(* CODESYS project pp-csp-handover-v4.project

Project tree, tasks and I/O mapping:
  PLC : HX-CP1S08, Hitachi Industrial Equipment Systems Co., Ltd., order no. HX-CP1S08, version 3.5.8.24
      settings: IP Address = '192.168.137.20'
    application Application
      libraries: Unit Conversion Interfaces, * (Intern); Standard, * (System); VisuDialogs, * (System); CAA Device Diagnosis, 3.5.4.0 (CAA Technical Workgroup); CAA Net Base Services, 3.5.8.10 (CAA Technical Workgroup); NetVarUdp, 3.5.17.0 (System); PRO JSON, 1.0.0.13 (Pro Electric)
      task VISU_TASK (cyclic, interval 200 ms, priority 31) calls VisuElems.Visu_Prg
      task EtherCAT_Task (cyclic, interval 4 ms, priority 1) calls CSP_Cycle, CSP_WriteOutputs
      task Task (cyclic, interval 5 ms, priority 5) calls main, TcpClient
      global variables gvlSetting
      data type ServoData
      program TcpClient [ST]
      program main [ST]
      visualisation Main
      global variables GVL
      program DriveDiagnostics [ST]
      function AppendDiagnosticText [ST]
      function BuildDiagnosticFeedback [ST]
      function LongStringLength [ST]
      data type CSP_AxisData
      function CSP_Bezier [ST]
      function block CSP_Brake [ST]
      global variables CSP_Config
      program CSP_Cycle [ST]
      global variables CSP_Data
      function CSP_Feedback [ST]
      function CSP_ParseFrame [ST]
      function CSP_ReadAxis [ST]
      function CSP_ReadNumber [ST]
      function block CSP_Receive [ST]
      function block CSP_Trajectory6 [ST]
      function CSP_WriteAxis [ST]
      program CSP_WriteOutputs [ST]
      data type PlatformControlState
      program PlatformStartup [ST]
      function CSP_StopOffset [ST]
    Basic : Basic, Hitachi-IES, version 3.5.8.20
      _16_Digital_Input : 16 Digital Input, Hitachi-IES, version 3.4.0.0
          input  Application.GVL.resetButton : BOOL  // ReserveWord0Type.Bit1
          input  Application.GVL.startButton : BOOL  // ReserveWord0Type.Bit2
          input  Application.GVL.stopButton : BOOL  // ReserveWord0Type.Bit3
          input  Application.GVL.safetySystem : BOOL  // ReserveWord0Type.Bit4
          unmapped channels: ReserveWord0Type, ReserveWord0Type, ReserveWord0Type
      _16_Digital_Output : 16 Digital Output, Hitachi-IES, version 3.4.0.0
          output Application.GVL.LightGreen : BOOL  // ReserveWord0Type.Bit0
          output Application.GVL.LightYellow : BOOL  // ReserveWord0Type.Bit1
          output Application.GVL.LightRed : BOOL  // ReserveWord0Type.Bit2
          unmapped channels: ReserveWord0Type, ReserveWord0Type, ReserveWord0Type
      <Empty>
      <Empty>
      _16_Digital_Input_1 : 16 Digital Input, Hitachi-IES, version 3.4.0.0
          unmapped channels: ReserveWord0Type, ReserveWord0Type, ReserveWord0Type
      <Empty>
      <Empty>
      <Empty>
      <Empty>
      <Empty>
      _16_Digital_Output_1 : 16 Digital Output, Hitachi-IES, version 3.4.0.0
          unmapped channels: ReserveWord0Type, ReserveWord0Type, ReserveWord0Type
    EtherCAT_Master : EtherCAT Master, Festo, version 3.5.16.43
        settings: MasterCycleTime = 4000; MasterUseLRW = False; SlaveAutoRestart = True; NetworkName = 'eth2'; NetworkName = "eth2"; SelectNetworkByName = False; EnableTaskMessage = False; SrcAddress1 = 42135; SrcAddress2 = 3137775364; EnableSecondAdapter = False; SrcAddress = [16#A4,16#97,16#BB,16#06,16#A7,16#04]; NetworkName = 'eth2'; NetworkName = "eth2"; SelectNetworkByName = False
      servo_drive_4 : CMMT-AS (FlightSim PP/CSP), Festo, order no. 5340819, 534082x, 813335x, version 1.0.0.0
          settings: Watchdog register 0400 = 2498; Watchdog register 0410 = 3000; Watchdog register 0420 = 1000; Physical Address of the Slave = 1002; AutoIncr Address of the Slave = 4294967295; FMMU.Global Start Address = 16#02000018; FMMU.Physical Start Address = 16#1000; FMMU.Access = 16#02; FMMU.Global Start Address = 16#01000012; FMMU.Physical Start Address = 16#1100; FMMU.Access = 16#01; FMMU.Global Start Address = 16#00080000; FMMU.StartBit = 1; FMMU.EndBit = 1; FMMU.Physical Start Address = 16#080D; FMMU.Access = 16#01; DC sync0 cycletime = 4000; DC enable = 1; DC sync0 enable = 1; DC sync1 cycletime = 4000; DC sync1 enable = 0
          unmapped channels: Controlword, Modes of operation, Target position, Profile velocity, Target velocity, Target torque, Velocity offset, Torque offset, ---, Statusword, Modes of operation display, Position actual value, Velocity actual value, Torque actual value, Multiturns actual value, ---
      servo_drive_3 : CMMT-AS (FlightSim PP/CSP), Festo, order no. 5340819, 534082x, 813335x, version 1.0.0.0
          settings: Watchdog register 0400 = 2498; Watchdog register 0410 = 3000; Watchdog register 0420 = 1000; Physical Address of the Slave = 1002; AutoIncr Address of the Slave = 4294967295; FMMU.Global Start Address = 16#02000018; FMMU.Physical Start Address = 16#1000; FMMU.Access = 16#02; FMMU.Global Start Address = 16#01000012; FMMU.Physical Start Address = 16#1100; FMMU.Access = 16#01; FMMU.Global Start Address = 16#00080000; FMMU.StartBit = 1; FMMU.EndBit = 1; FMMU.Physical Start Address = 16#080D; FMMU.Access = 16#01; DC sync0 cycletime = 4000; DC enable = 1; DC sync0 enable = 1; DC sync1 cycletime = 4000; DC sync1 enable = 0
          unmapped channels: Controlword, Modes of operation, Target position, Profile velocity, Target velocity, Target torque, Velocity offset, Torque offset, ---, Statusword, Modes of operation display, Position actual value, Velocity actual value, Torque actual value, Multiturns actual value, ---
      servo_drive_2 : CMMT-AS (FlightSim PP/CSP), Festo, order no. 5340819, 534082x, 813335x, version 1.0.0.0
          settings: Watchdog register 0400 = 2498; Watchdog register 0410 = 3000; Watchdog register 0420 = 1000; Physical Address of the Slave = 1002; AutoIncr Address of the Slave = 4294967295; FMMU.Global Start Address = 16#02000018; FMMU.Physical Start Address = 16#1000; FMMU.Access = 16#02; FMMU.Global Start Address = 16#01000012; FMMU.Physical Start Address = 16#1100; FMMU.Access = 16#01; FMMU.Global Start Address = 16#00080000; FMMU.StartBit = 1; FMMU.EndBit = 1; FMMU.Physical Start Address = 16#080D; FMMU.Access = 16#01; DC sync0 cycletime = 4000; DC enable = 1; DC sync0 enable = 1; DC sync1 cycletime = 4000; DC sync1 enable = 0
          unmapped channels: Controlword, Modes of operation, Target position, Profile velocity, Target velocity, Target torque, Velocity offset, Torque offset, ---, Statusword, Modes of operation display, Position actual value, Velocity actual value, Torque actual value, Multiturns actual value, ---
      servo_drive_1 : CMMT-AS (FlightSim PP/CSP), Festo, order no. 5340819, 534082x, 813335x, version 1.0.0.0
          settings: Watchdog register 0400 = 2498; Watchdog register 0410 = 3000; Watchdog register 0420 = 1000; Physical Address of the Slave = 1001; FMMU.Global Start Address = 16#02000000; FMMU.Physical Start Address = 16#1000; FMMU.Access = 16#02; FMMU.Global Start Address = 16#01000000; FMMU.Physical Start Address = 16#1100; FMMU.Access = 16#01; FMMU.Global Start Address = 16#00080000; FMMU.Physical Start Address = 16#080D; FMMU.Access = 16#01; DC sync0 cycletime = 4000; DC enable = 1; DC sync0 enable = 1; DC sync1 cycletime = 4000; DC sync1 enable = 0
          unmapped channels: Controlword, Modes of operation, Target position, Profile velocity, Target velocity, Target torque, Velocity offset, Torque offset, ---, Statusword, Modes of operation display, Position actual value, Velocity actual value, Torque actual value, Multiturns actual value, ---
      servo_drive_6 : CMMT-AS (FlightSim PP/CSP), Festo, order no. 5340819, 534082x, 813335x, version 1.0.0.0
          settings: Watchdog register 0400 = 2498; Watchdog register 0410 = 3000; Watchdog register 0420 = 1000; Physical Address of the Slave = 1002; AutoIncr Address of the Slave = 4294967295; FMMU.Global Start Address = 16#02000018; FMMU.Physical Start Address = 16#1000; FMMU.Access = 16#02; FMMU.Global Start Address = 16#01000012; FMMU.Physical Start Address = 16#1100; FMMU.Access = 16#01; FMMU.Global Start Address = 16#00080000; FMMU.StartBit = 1; FMMU.EndBit = 1; FMMU.Physical Start Address = 16#080D; FMMU.Access = 16#01; DC sync0 cycletime = 4000; DC enable = 1; DC sync0 enable = 1; DC sync1 cycletime = 4000; DC sync1 enable = 0
          unmapped channels: Controlword, Modes of operation, Target position, Profile velocity, Target velocity, Target torque, Velocity offset, Torque offset, ---, Statusword, Modes of operation display, Position actual value, Velocity actual value, Torque actual value, Multiturns actual value, ---
      servo_drive_5 : CMMT-AS (FlightSim PP/CSP), Festo, order no. 5340819, 534082x, 813335x, version 1.0.0.0
          settings: Watchdog register 0400 = 2498; Watchdog register 0410 = 3000; Watchdog register 0420 = 1000; Physical Address of the Slave = 1002; AutoIncr Address of the Slave = 4294967295; FMMU.Global Start Address = 16#02000018; FMMU.Physical Start Address = 16#1000; FMMU.Access = 16#02; FMMU.Global Start Address = 16#01000012; FMMU.Physical Start Address = 16#1100; FMMU.Access = 16#01; FMMU.Global Start Address = 16#00080000; FMMU.StartBit = 1; FMMU.EndBit = 1; FMMU.Physical Start Address = 16#080D; FMMU.Access = 16#01; DC sync0 cycletime = 4000; DC enable = 1; DC sync0 enable = 1; DC sync1 cycletime = 4000; DC sync1 enable = 0
          unmapped channels: Controlword, Modes of operation, Target position, Profile velocity, Target velocity, Target torque, Velocity offset, Torque offset, ---, Statusword, Modes of operation display, Position actual value, Velocity actual value, Torque actual value, Multiturns actual value, ---
  libraries: VisuSymbols, 4.1.0.0 (System)
  function block Axis [ST]: enabled, init, doAbort, isReady, doMovement, doReset, getPosition, inError, cycle, isInitialised, PPMoveDone
  function block signal [ST]: init, cycle
  text list GlobalTextList
  function block Light [ST]: blink, init, cycle, enable
  function block FlightSimulator [ST]: safetyStop, doReset, isEnabled, getPositions, cycle, goNeutralPosition, isReady, doMovement, isInitialised, init, inError, goHomePosition, goTopPosition, PPState
  data type stateFlightSimulator
*)

// PLC/Application/ServoData
TYPE ServoData :
STRUCT
	positions: ARRAY[1..6] OF JSONVAR;
	speeds: ARRAY[1..6] OF JSONVAR;
END_STRUCT
END_TYPE

// stateFlightSimulator
{attribute 'qualified_only'}
{attribute 'strict'}
TYPE stateFlightSimulator :
(
	error  := 0,
	resetting,
	stopped,
	starting,
	started,
	stopping
);
END_TYPE

// PLC/Application/CSP_AxisData
TYPE CSP_AxisData :
STRUCT
    RequestedPosition : LREAL;
    CommandPosition : LREAL;
    CommandVelocity : LREAL;
    CommandAcceleration : LREAL;
    ActualPosition : LREAL;
    ActualVelocity : LREAL;
    FollowingError : LREAL;
    PositionFactor : LREAL;
    VelocityFactor : LREAL;
    ActualRaw : DINT;
    TargetRaw : DINT;
    FollowingErrorRaw : DINT;
    ModeRequested : SINT;
    ModeActual : SINT;
    Statusword : WORD;
    Controlword : WORD;
    CiA402State : WORD;
    PositionLimit : BOOL;
    CommunicationTimeout : BOOL;
    Ready : BOOL;
    // 0 ready; 1 PDO pointer; 2 SDO init; 3 factor; 4 bus; 5 conversion mismatch.
    ReadinessCode : UINT;
    VelocityAllowed : LREAL;
END_STRUCT
END_TYPE

// PLC/Application/PlatformControlState
{attribute 'qualified_only'}
{attribute 'strict'}
TYPE PlatformControlState :
(
    PP_RESET := 0,
    PP_STOPPED := 1,
    PP_STARTING := 2,
    CSP_HANDOVER := 3,
    CSP_READY := 4,
    CSP_RUNNING := 5,
    CSP_RECOVERY := 6,
    FAULT := 7,
    PP_HANDBACK := 8 // Reset: CSP brakes and restores mode 1, then PP resumes
);
END_TYPE

// PLC/Application/gvlSetting
{attribute 'qualified_only'}
VAR_GLOBAL CONSTANT
    // Port to use to send data.
	gc_uiPort        : UINT := 32760;
    // IP Address of the computer that hosts the software.
	gc_stIpAddr      : NBS.IP_ADDR := (sAddr := '192.168.137.123');
	// Length of the telegram.
    gc_wMaxTelegram  : INT := 512;
END_VAR

// PLC/Application/GVL
{attribute 'qualified_only'}
VAR_GLOBAL
	// Red light on electrical housing.
	lightRed: BOOL;
	// Yellow light on electrical housing.
	lightYellow: BOOL;
	// Green light on electrical housing.
	lightGreen: BOOL;
	// Reset button on electrical housing.
	resetButton: BOOL := FALSE;
	// Start button on electrical housing.
	startButton: BOOL := FALSE;
	// Stop button on electrical housing.
	stopButton: BOOL := FALSE;
	// Safety system, connected to safety relay.
	safetySystem: BOOL := FALSE;
	// Virtual reset button on HMI.
	resetHMI: BOOL;
	// Virtual start button on HMI.
	startHMI: BOOL;
	// Virtual stop button on HMI.
	stopHMI: BOOL;
	// Virtual toggle button to toggle between tCP data and manual data on HMI.
	useTCPData: BOOL := TRUE;
	// Manual slider velocity input on HMI.
	nextVelocityInput: REAL := 200;
	// Manual slider position input on HMI.
	nextPositionInput: REAL := 0;
	// Flight simulator object.
	FlightSimulator: FlightSimulator;
	// Velocity input from TCP data or HMI data.
	servoVelocities: ARRAY[1..6] OF REAL;
	// Position input from TCP data or HMI data.
	servoPositions: ARRAY[1..6] OF REAL;
	// Current Positions in array format.
	servoPositionsCurrent: ARRAY[1..6] OF REAL;
	// Current Positions in JSON format, used to send back to TCP client.
	currentPositions: ARRAY[1..6] OF JSONVAR;
END_VAR

// PLC/Application/CSP_Config
{attribute 'qualified_only'}
VAR_GLOBAL CONSTANT
    CONTROL_MODE_PP : SINT := 1;
    CONTROL_MODE_CSP : SINT := 8;
    // Match BuildMode.h. PP remains the initial commissioning selection.
    ControlMode : SINT := 8;
    // Also set EtherCAT_Task, master cycle and slave DC Sync0 to this interval.
    CycleSeconds : LREAL := 0.004;
    MinimumPosition : LREAL := 10.0;
    MaximumPosition : LREAL := 390.0;
    MaximumVelocity : LREAL := 100; // mm/s; commissioning starting values
    MaximumAcceleration : LREAL := 200; // mm/s^2
    BrakingAcceleration : LREAL := 200; // <= MaximumAcceleration
    MaximumJerk : LREAL := 1000; // mm/s^3
    CommunicationTimeout : TIME := T#500MS;
    TransitionTimeout : TIME := T#10S;
    StandstillVelocity : LREAL := 0.05;
    HomePosition : LREAL := 200.0;
    HomeTolerance : LREAL := 0.5;
    HomeSettleTime : TIME := T#200MS;
    HomeTimeout : TIME := T#60S;
    // Set TRUE only after the eight required PDOs, DC, interpolation period,
    // actual task timing and all six existing position conversions are checked.
    Commissioned : BOOL := TRUE;
END_VAR

// PLC/Application/CSP_Data
{attribute 'qualified_only'}
VAR_GLOBAL
    Axis : ARRAY[1..6] OF CSP_AxisData;
    CycleCounter : UDINT;
    // TCP writes odd generation, complete target, then even generation. The
    // higher-priority motion task only accepts matching even generations.
    Generation : UDINT;
    ReceivedPosition : ARRAY[1..6] OF LREAL;
    ReceivedMode : SINT;
    ReceivedTick : UDINT;
    Connected : BOOL;
    Enable : BOOL;
    Reset : BOOL;
    StopRequested : BOOL;
    ResetRequired : BOOL := TRUE;
    Homing : BOOL; // park at HomePosition using the existing encoder reference
    ReadyToStart : BOOL;
    OwnsOutputs : BOOL; // FALSE: vendor PP writer; TRUE: direct CSP writer
    PlatformState : PlatformControlState := PlatformControlState.PP_RESET;
    PPReleased : BOOL; // published by PP task only after its last complete call
    // Published by the CSP task only after it restored mode 1 and stopped writing.
    // PP clears PPReleased in response; CSP then clears this flag.
    CSPReleased : BOOL;
    PPMoveDone : ARRAY[1..6] OF BOOL;
    AllPPMoveDone, AllStationary, AllCSPModeConfirmed : BOOL;
    // The exact PP-side handover condition, evaluated in the PP task.
    PPStartupComplete : BOOL;
    // First axis whose mode display differs from the requested handover mode
    // (8 during CSP_HANDOVER, 1 during PP_HANDBACK); 0 = all confirmed.
    ModeBlockingAxis : INT;
    InitialTargetRaw : ARRAY[1..6] OF DINT;
    // FaultCode that Reset acknowledged before ownership returned to PP.
    LastCSPFaultCode : UINT;
    Active : BOOL;
    TransitionState : UINT;
    Fault : BOOL;
    FaultCode : UINT;
    // Frozen at timeout, before quick stop changes the live drive states.
    TimeoutState : UINT;
    TimeoutStatusword : ARRAY[1..6] OF WORD;
    TimeoutControlword : ARRAY[1..6] OF WORD;
    // 0 running/transitioning; 1 commissioning; 2 axis readiness; 3 safety;
    // 4 operator Start; 5 fresh PC target; 6 drive mode; 7 fault (see FaultCode).
    // While PP owns the drives: 10 PP not in STARTED; 11 not stationary;
    // 12 PP move still executing / no drive Standstill (FlightSimulator.isReady);
    // 13 an axis is outside HomeTolerance of HomePosition; 14 MC_MoveAbsolute
    // Error/CommandAborted. PPMoveDone[1..6] shows the axis.
    StartupBlockReason : UINT;
    ReversalDeferred : BOOL;
    // Map 0x60F4:00 (DINT) from each drive here; not computed PC error.
    FollowingErrorRaw : ARRAY[1..6] OF DINT;
END_VAR

// PLC/Application/CSP_Cycle
PROGRAM CSP_Cycle
VAR
    trajectory : CSP_Trajectory6;
    actual, requested, receivedCopy : ARRAY[1..6] OF LREAL;
    generation, generationAfter, acceptedGeneration, tick : UDINT;
    packetMode : SINT;
    packetTick, receivedTickCopy : UDINT;
    newTarget, timedOut, allReady, allStopped, allDisabled, allMode, allEnabled, allSwitchedOn, allPPMode : BOOL;
    resetEdge : R_TRIG;
    resetRequest : BOOL;
    resetConditionsReady, anyDriveFaultReaction : BOOL;
    standstill : TON;
    transition : TON;
    previousTransitionState : UINT;
    homePhase : UINT; // 1 brake, 2 plan park move, 3 wait for measured arrival
    homeTarget : ARRAY[1..6] OF LREAL;
    homeSettled, homeTimer : TON;
    homeAtPosition : BOOL;
    handoverValid : BOOL;
    initialPosition : ARRAY[1..6] OF LREAL; // captured at the PP -> CSP ownership switch
    holdRaw : ARRAY[1..6] OF DINT; // stationary target while restoring PP mode
    expectedMode : SINT;
    i : INT;
    stateWord : WORD;
    distance : LREAL;
END_VAR

IF CSP_Config.ControlMode <> CSP_Config.CONTROL_MODE_CSP THEN RETURN; END_IF
CSP_Data.CycleCounter := CSP_Data.CycleCounter+1;
CSP_ReadAxis(Axis:=servo_drive_1,PlatformAxis:=1);
CSP_ReadAxis(Axis:=servo_drive_2,PlatformAxis:=2);
CSP_ReadAxis(Axis:=servo_drive_3,PlatformAxis:=3);
CSP_ReadAxis(Axis:=servo_drive_4,PlatformAxis:=4);
CSP_ReadAxis(Axis:=servo_drive_5,PlatformAxis:=5);
CSP_ReadAxis(Axis:=servo_drive_6,PlatformAxis:=6);
tick := TIME_TO_UDINT(TIME());
resetEdge(CLK:=CSP_Data.Reset);
IF resetEdge.Q THEN
    resetRequest := TRUE;
END_IF;
newTarget := FALSE;
generation := CSP_Data.Generation;
IF generation MOD 2 = 0 AND generation <> acceptedGeneration THEN
    receivedCopy := CSP_Data.ReceivedPosition;
    packetMode := CSP_Data.ReceivedMode; receivedTickCopy := CSP_Data.ReceivedTick;
    generationAfter := CSP_Data.Generation;
    IF generation = generationAfter AND packetMode = 8 THEN
        acceptedGeneration := generation; newTarget := TRUE;
        requested := receivedCopy; packetTick := receivedTickCopy;

    END_IF
END_IF
timedOut := NOT CSP_Data.Connected OR acceptedGeneration = 0
    OR (tick - packetTick) > TIME_TO_UDINT(CSP_Config.CommunicationTimeout);
allReady := TRUE; allStopped := TRUE; allDisabled := TRUE; allMode := TRUE; allEnabled := TRUE; allSwitchedOn := TRUE;
allPPMode := TRUE;
FOR i := 1 TO 6 DO
    stateWord := CSP_Data.Axis[i].Statusword AND 16#006F;
    CSP_Data.Axis[i].CiA402State := stateWord;
    actual[i] := CSP_Data.Axis[i].ActualPosition;
    allReady := allReady AND CSP_Data.Axis[i].Ready;
    allStopped := allStopped AND ABS(CSP_Data.Axis[i].ActualVelocity) <= CSP_Config.StandstillVelocity;
    allDisabled := allDisabled AND (stateWord = 16#0023 OR stateWord = 16#0021 OR (stateWord AND 16#004F) = 16#0040);
    allMode := allMode AND CSP_Data.Axis[i].ModeActual = 8;
    allPPMode := allPPMode AND CSP_Data.Axis[i].ModeActual = CSP_Config.CONTROL_MODE_PP;
    allEnabled := allEnabled AND stateWord = 16#0027;
    allSwitchedOn := allSwitchedOn AND (stateWord = 16#0023 OR stateWord = 16#0027);
    CSP_Data.Axis[i].CommunicationTimeout := timedOut;
    CSP_Data.Axis[i].PositionLimit := CSP_Data.Axis[i].RequestedPosition < CSP_Config.MinimumPosition
        OR CSP_Data.Axis[i].RequestedPosition > CSP_Config.MaximumPosition;
END_FOR
// Read-only monitoring runs during PP startup; no CSP output ownership yet.
standstill(IN:=allReady AND allStopped, PT:=T#200MS);
CSP_Data.AllStationary := standstill.Q;
CSP_Data.AllCSPModeConfirmed := allMode;
// Mode the drives must display for the current owner; first mismatch is exposed.
IF CSP_Data.OwnsOutputs AND CSP_Data.TransitionState < 70 THEN expectedMode := 8;
ELSE expectedMode := CSP_Config.CONTROL_MODE_PP; END_IF
CSP_Data.ModeBlockingAxis := 0;
FOR i := 6 TO 1 BY -1 DO
    IF CSP_Data.Axis[i].ModeActual <> expectedMode THEN CSP_Data.ModeBlockingAxis := i; END_IF
END_FOR
// PP acknowledged the Reset handback by withdrawing PPReleased.
IF CSP_Data.CSPReleased AND NOT CSP_Data.PPReleased THEN CSP_Data.CSPReleased := FALSE; END_IF
IF NOT CSP_Data.OwnsOutputs THEN
    // PP owns Reset while it owns the drives; do not replay its edges later.
    IF NOT CSP_Data.PPReleased THEN resetRequest := FALSE; END_IF
    IF CSP_Data.PPReleased AND NOT CSP_Data.CSPReleased THEN
        // The slower PP task published this only AFTER its last motion call.
        // Capture all axes before atomically selecting the sole CSP writer.
        handoverValid := CSP_Config.CycleSeconds > 0 AND CSP_Config.MaximumVelocity > 0
            AND CSP_Config.MaximumAcceleration > 0 AND CSP_Config.BrakingAcceleration > 0
            AND CSP_Config.BrakingAcceleration <= CSP_Config.MaximumAcceleration
            AND CSP_Config.MaximumJerk > 0 AND CSP_Config.MinimumPosition < CSP_Config.MaximumPosition;
        FOR i := 1 TO 6 DO
            handoverValid := handoverValid AND actual[i] >= CSP_Config.MinimumPosition
                AND actual[i] <= CSP_Config.MaximumPosition AND CSP_Data.Axis[i].ModeActual = 1;
            // Bumpless transfer: the first CSP target is the measured raw position.
            CSP_Data.InitialTargetRaw[i] := CSP_Data.Axis[i].ActualRaw;
            initialPosition[i] := actual[i]; // = ActualRaw * PositionFactor
            CSP_Data.Axis[i].TargetRaw := CSP_Data.InitialTargetRaw[i];
            CSP_Data.Axis[i].RequestedPosition := initialPosition[i];
            CSP_Data.Axis[i].CommandPosition := initialPosition[i];
            CSP_Data.Axis[i].CommandVelocity := 0;
            CSP_Data.Axis[i].CommandAcceleration := 0;
            CSP_Data.Axis[i].ModeRequested := 8;
            CSP_Data.Axis[i].Controlword := 16#000F;
        END_FOR
        CSP_Data.Active := FALSE; CSP_Data.ReadyToStart := FALSE;
        CSP_Data.Homing := FALSE; homePhase := 0;
        // A Reset edge seen in this capture window is kept: it returns to PP.
        CSP_Data.TransitionState := 60;
        previousTransitionState := 0;
        transition(IN:=FALSE, PT:=CSP_Config.TransitionTimeout);
        CSP_Data.PlatformState := PlatformControlState.CSP_HANDOVER;
        // Stop/Reset here are not faults: CSP holds, and Reset hands back to PP.
        IF NOT allReady OR NOT standstill.Q OR NOT allEnabled OR NOT GVL.safetySystem
            OR NOT CSP_Config.Commissioned OR NOT handoverValid OR CSP_Data.Fault THEN
            CSP_Data.Fault := TRUE; CSP_Data.FaultCode := 10;
            CSP_Data.PlatformState := PlatformControlState.FAULT;
            FOR i := 1 TO 6 DO
                CSP_Data.Axis[i].Controlword := 16#0002;
                CSP_Data.Axis[i].ModeRequested := CSP_Data.Axis[i].ModeActual;
            END_FOR
        END_IF
        CSP_Data.OwnsOutputs := TRUE; // sole ownership switch, in EtherCAT task
    END_IF
    RETURN;
END_IF
homeAtPosition := TRUE;
FOR i := 1 TO 6 DO
    homeTarget[i] := CSP_Config.HomePosition;
    homeAtPosition := homeAtPosition AND ABS(actual[i]-CSP_Config.HomePosition) <= CSP_Config.HomeTolerance;
END_FOR
homeSettled(IN:=CSP_Data.Homing AND homePhase = 3 AND NOT trajectory.Busy
    AND homeAtPosition AND allReady AND allStopped, PT:=CSP_Config.HomeSettleTime);
homeTimer(IN:=CSP_Data.Homing AND NOT CSP_Data.Fault, PT:=CSP_Config.HomeTimeout);
IF homeTimer.Q AND NOT CSP_Data.Fault THEN
    CSP_Data.Fault := TRUE; CSP_Data.FaultCode := 8;
END_IF
CSP_Data.StartupBlockReason := 0;
IF CSP_Data.Fault THEN CSP_Data.StartupBlockReason := 7;
ELSIF NOT CSP_Config.Commissioned THEN CSP_Data.StartupBlockReason := 1;
ELSIF NOT allReady THEN CSP_Data.StartupBlockReason := 2;
ELSIF NOT GVL.safetySystem THEN CSP_Data.StartupBlockReason := 3;
ELSIF CSP_Data.Homing THEN CSP_Data.StartupBlockReason := 9;
ELSIF CSP_Data.ResetRequired THEN CSP_Data.StartupBlockReason := 8;
ELSIF NOT CSP_Data.Enable THEN CSP_Data.StartupBlockReason := 4;
ELSIF timedOut THEN CSP_Data.StartupBlockReason := 5;
ELSIF NOT allMode THEN CSP_Data.StartupBlockReason := 6;
END_IF
// Each transition gets a fresh timeout. A latched fault must stop/reset
// the TON; otherwise Reset -> state 20 immediately faults again on old Q.
transition(IN:=NOT CSP_Data.Fault
    AND CSP_Data.TransitionState = previousTransitionState
    AND ((CSP_Data.TransitionState > 0 AND CSP_Data.TransitionState < 40)
        OR (CSP_Data.TransitionState = 40 AND CSP_Data.Homing)
        OR CSP_Data.TransitionState = 60 OR CSP_Data.TransitionState >= 70),
    PT:=CSP_Config.TransitionTimeout);
previousTransitionState := CSP_Data.TransitionState;
IF transition.Q AND NOT CSP_Data.Fault THEN
    CSP_Data.TimeoutState := CSP_Data.TransitionState;
    FOR i := 1 TO 6 DO
        CSP_Data.TimeoutStatusword[i] := CSP_Data.Axis[i].Statusword;
        CSP_Data.TimeoutControlword[i] := CSP_Data.Axis[i].Controlword;
    END_FOR
    CSP_Data.Fault := TRUE; CSP_Data.FaultCode := 1;
END_IF
// Keep the first cause latched; later consequences must not overwrite it.
IF NOT CSP_Data.Fault AND CSP_Data.OwnsOutputs AND (NOT allReady OR NOT GVL.safetySystem) THEN
    CSP_Data.Fault := TRUE; CSP_Data.FaultCode := 2;
END_IF
IF CSP_Data.Fault THEN
    CSP_Data.PlatformState := PlatformControlState.FAULT;
    CSP_Data.Active := FALSE;
    CSP_Data.ResetRequired := TRUE; CSP_Data.ReadyToStart := FALSE;
    CSP_Data.Homing := FALSE; homePhase := 0;
    anyDriveFaultReaction := FALSE;
    FOR i := 1 TO 6 DO
        CSP_Data.Axis[i].Controlword := 16#0002;
        anyDriveFaultReaction := anyDriveFaultReaction
            OR (CSP_Data.Axis[i].Statusword AND 16#004F) = 16#000F;
    END_FOR
    resetConditionsReady := standstill.Q AND GVL.safetySystem AND allReady
        AND NOT CSP_Data.Enable AND NOT CSP_Data.StopRequested AND CSP_Config.Commissioned;
    // Reset returns the drives to the original PP reset (MC_Reset_Festo etc.).
    // CSP issues no CiA402 fault-reset pulse itself; a drive in Fault stays
    // quick-stopped/disabled while its mode display is restored to 1.
    IF resetRequest AND resetConditionsReady AND NOT anyDriveFaultReaction THEN
        transition(IN:=FALSE, PT:=CSP_Config.TransitionTimeout);
        previousTransitionState := 0;
        CSP_Data.LastCSPFaultCode := CSP_Data.FaultCode;
        CSP_Data.Fault := FALSE; CSP_Data.FaultCode := 0;
        CSP_Data.TransitionState := 70;
        CSP_Data.PlatformState := PlatformControlState.PP_HANDBACK;
        resetRequest := FALSE;
    END_IF
    RETURN;
END_IF
// Reset belongs to the original PP state machine. A Reset during CSP handover
// or operation first brakes the existing command continuously (state 70), then
// restores mode 1 (state 71) and releases the drives to PP. States 0..40 and
// the CSP park move are not entered under this PP-startup policy.
IF resetRequest AND CSP_Data.TransitionState >= 50 AND CSP_Data.TransitionState < 70 THEN
    CSP_Data.ResetRequired := TRUE; CSP_Data.ReadyToStart := FALSE;
    CSP_Data.TransitionState := 70;
    resetRequest := FALSE;
END_IF
IF CSP_Data.StopRequested AND CSP_Data.Homing THEN
    CSP_Data.Homing := FALSE; homePhase := 0;
    CSP_Data.ResetRequired := TRUE; CSP_Data.ReadyToStart := FALSE;
END_IF
IF CSP_Data.Homing AND (CSP_Config.HomePosition < CSP_Config.MinimumPosition
    OR CSP_Config.HomePosition > CSP_Config.MaximumPosition OR CSP_Config.HomeTolerance <= 0
    OR CSP_Config.HomeTimeout <= T#0MS OR CSP_Config.HomeSettleTime <= T#0MS) THEN
    CSP_Data.Homing := FALSE; CSP_Data.Fault := TRUE; CSP_Data.FaultCode := 3; RETURN;
END_IF
CASE CSP_Data.TransitionState OF
60:
    // PP already enabled and positioned every axis. Do not disable/re-enable.
    // Hold the captured positions while changing mode; no PC targets are consumed.
    // A drive that leaves operation-enabled or moves away aborts the handover.
    handoverValid := allEnabled;
    FOR i := 1 TO 6 DO
        handoverValid := handoverValid
            AND ABS(actual[i]-initialPosition[i]) <= CSP_Config.HomeTolerance;
    END_FOR
    IF NOT handoverValid THEN
        CSP_Data.Fault := TRUE; CSP_Data.FaultCode := 10;
        FOR i := 1 TO 6 DO CSP_Data.Axis[i].Controlword := 16#0002; END_FOR
        RETURN;
    END_IF
    FOR i := 1 TO 6 DO
        CSP_Data.Axis[i].TargetRaw := CSP_Data.InitialTargetRaw[i];
        CSP_Data.Axis[i].CommandPosition := initialPosition[i];
        CSP_Data.Axis[i].RequestedPosition := initialPosition[i];
        CSP_Data.Axis[i].ModeRequested := 8;
        CSP_Data.Axis[i].Controlword := 16#000F;
    END_FOR
    // All-six barrier: the platform stays in handover until every display is 8.
    IF allMode THEN
        trajectory(Initialize:=TRUE, Actual:=initialPosition);
        CSP_Data.Active := TRUE; CSP_Data.ReadyToStart := TRUE;
        CSP_Data.ResetRequired := FALSE;
        CSP_Data.PlatformState := PlatformControlState.CSP_READY;
        CSP_Data.TransitionState := 61;
        // Hold for another whole cycle; earlier/cached network targets ignored.
    END_IF
61:
    IF NOT allMode OR NOT allEnabled THEN
        CSP_Data.Fault := TRUE; CSP_Data.FaultCode := 6;
        FOR i := 1 TO 6 DO CSP_Data.Axis[i].Controlword := 16#0002; END_FOR
        RETURN;
    END_IF
    CSP_Data.TransitionState := 50;
    // No trajectory update in this cycle. Only a later valid packet can move.
0:
    // Remain reset-required until the operator explicitly requests the park move.
    IF CSP_Data.Homing AND CSP_Config.Commissioned AND allReady AND GVL.safetySystem THEN
        IF CSP_Config.CycleSeconds <= 0 OR CSP_Config.MaximumVelocity <= 0
            OR CSP_Config.MaximumAcceleration <= 0 OR CSP_Config.BrakingAcceleration <= 0
            OR CSP_Config.BrakingAcceleration > CSP_Config.MaximumAcceleration
            OR CSP_Config.MaximumJerk <= 0 OR CSP_Config.MinimumPosition >= CSP_Config.MaximumPosition THEN
            CSP_Data.Fault := TRUE; CSP_Data.FaultCode := 3; RETURN;
        END_IF
        FOR i := 1 TO 6 DO
            CSP_Data.Axis[i].TargetRaw := CSP_Data.Axis[i].ActualRaw;
            CSP_Data.Axis[i].ModeRequested := CSP_Data.Axis[i].ModeActual;
            IF CSP_Data.Axis[i].CiA402State = 16#0027 THEN CSP_Data.Axis[i].Controlword := 16#010F;
            ELSE CSP_Data.Axis[i].Controlword := 16#0006; END_IF
        END_FOR
        CSP_Data.OwnsOutputs := TRUE; CSP_Data.TransitionState := 10;
    END_IF
10:
    // HALT in the current PP mode, retaining drive-configured PP deceleration.
    // Never switch mode or discard the moving setpoint before actual standstill.
    FOR i := 1 TO 6 DO
        IF CSP_Data.Axis[i].CiA402State = 16#0027 THEN
            CSP_Data.Axis[i].Controlword := 16#010F;
        ELSE CSP_Data.Axis[i].Controlword := 16#0006;
        END_IF
    END_FOR
    IF standstill.Q THEN CSP_Data.TransitionState := 20; END_IF
20:
    FOR i := 1 TO 6 DO
        CSP_Data.Axis[i].Controlword := 16#0007; // disable operation, retain voltage
        IF CSP_Data.Axis[i].CiA402State = 16#0007 THEN
            CSP_Data.Axis[i].Controlword := 0; // leave quick-stop-active via disable voltage
        END_IF
        CSP_Data.Axis[i].TargetRaw := CSP_Data.Axis[i].ActualRaw;
    END_FOR
    IF allDisabled THEN CSP_Data.TransitionState := 30; END_IF
30,40:
    FOR i := 1 TO 6 DO
        IF actual[i] < CSP_Config.MinimumPosition OR actual[i] > CSP_Config.MaximumPosition THEN
            CSP_Data.Fault := TRUE; CSP_Data.FaultCode := 5; RETURN;
        END_IF
    END_FOR
    FOR i := 1 TO 6 DO
        CSP_Data.Axis[i].TargetRaw := CSP_Data.Axis[i].ActualRaw;
        CSP_Data.Axis[i].ModeRequested := 8;
        stateWord := CSP_Data.Axis[i].CiA402State;
        CASE stateWord OF
            16#0040,16#0060: CSP_Data.Axis[i].Controlword := 16#0006;
            16#0021: CSP_Data.Axis[i].Controlword := 16#0007;
            16#0023,16#0027:
                CSP_Data.Axis[i].Controlword := 16#0007;
                // All-six mode barrier before ANY axis enables operation.
                IF allMode AND allSwitchedOn AND CSP_Data.Homing AND NOT CSP_Data.StopRequested THEN
                    CSP_Data.Axis[i].Controlword := 16#000F;
                END_IF
        ELSE
            CSP_Data.Axis[i].Controlword := 0;
            IF (stateWord AND 16#004F) = 16#0008 THEN CSP_Data.Fault := TRUE; CSP_Data.FaultCode := 4; END_IF
        END_CASE
    END_FOR
    IF allMode THEN CSP_Data.TransitionState := 40; END_IF
    IF allMode AND allEnabled AND CSP_Data.Homing AND NOT CSP_Data.StopRequested THEN
        FOR i := 1 TO 6 DO
            IF actual[i] < CSP_Config.MinimumPosition OR actual[i] > CSP_Config.MaximumPosition THEN
                CSP_Data.Fault := TRUE; CSP_Data.FaultCode := 5; RETURN;
            END_IF
        END_FOR
        trajectory(Initialize:=TRUE, Actual:=actual);
        FOR i := 1 TO 6 DO
            CSP_Data.Axis[i].CommandPosition := actual[i];
            CSP_Data.Axis[i].CommandVelocity := 0;
            CSP_Data.Axis[i].CommandAcceleration := 0;
        END_FOR
        CSP_Data.TransitionState := 50; CSP_Data.Active := TRUE;
        // Local park motion runs first; PC commands remain gated until a later Start.
    END_IF
50:
    IF NOT allMode OR NOT allEnabled THEN
        CSP_Data.Fault := TRUE; CSP_Data.FaultCode := 6; RETURN;
    END_IF
    IF CSP_Data.Homing THEN
        FOR i := 1 TO 6 DO CSP_Data.Axis[i].RequestedPosition := homeTarget[i]; END_FOR
        CASE homePhase OF
        1:
            trajectory(Initialize:=FALSE, NewTarget:=FALSE, Stop:=TRUE);
            IF NOT trajectory.Busy AND standstill.Q THEN homePhase := 2; END_IF
        2:
            trajectory(Initialize:=FALSE, NewTarget:=TRUE, Stop:=FALSE, Requested:=homeTarget);
            homePhase := 3;
        3:
            trajectory(Initialize:=FALSE, NewTarget:=FALSE, Stop:=FALSE);
            IF homeSettled.Q AND NOT trajectory.Busy THEN
                CSP_Data.Homing := FALSE; homePhase := 0;
                CSP_Data.ResetRequired := FALSE; CSP_Data.ReadyToStart := TRUE;
            END_IF
        END_CASE
    ELSE
        // No queued PC move may run during reset-required or park hold.
        trajectory(Initialize:=FALSE,
            NewTarget:=newTarget AND CSP_Data.ReadyToStart AND CSP_Data.Enable,
            Stop:=timedOut OR NOT CSP_Data.Enable OR NOT CSP_Data.ReadyToStart
                OR CSP_Data.StopRequested, Requested:=requested);
        IF newTarget AND CSP_Data.ReadyToStart AND CSP_Data.Enable THEN
            FOR i := 1 TO 6 DO CSP_Data.Axis[i].RequestedPosition := requested[i]; END_FOR
        END_IF
    END_IF
    IF trajectory.Fault THEN CSP_Data.Fault := TRUE; CSP_Data.FaultCode := 7; RETURN; END_IF
    IF CSP_Data.Homing OR CSP_Data.ResetRequired THEN
        CSP_Data.PlatformState := PlatformControlState.CSP_RECOVERY;
    ELSIF CSP_Data.Enable AND NOT timedOut AND (newTarget OR CSP_Data.PlatformState = PlatformControlState.CSP_RUNNING) THEN
        CSP_Data.PlatformState := PlatformControlState.CSP_RUNNING;
    ELSE
        CSP_Data.PlatformState := PlatformControlState.CSP_READY;
    END_IF
    // Festo factor is user units per raw count: output is the inverse of readback.
    CSP_Data.ReversalDeferred := trajectory.Deferred;
    FOR i := 1 TO 6 DO
        CSP_Data.Axis[i].CommandPosition := trajectory.P[i];
        CSP_Data.Axis[i].CommandVelocity := trajectory.V[i];
        CSP_Data.Axis[i].CommandAcceleration := trajectory.A[i];
        CSP_Data.Axis[i].TargetRaw := LREAL_TO_DINT(trajectory.P[i]/CSP_Data.Axis[i].PositionFactor);
        CSP_Data.Axis[i].Controlword := 16#000F; // only while operation-enabled in CSP
        IF trajectory.V[i] >= 0 THEN distance := CSP_Config.MaximumPosition-trajectory.P[i];
        ELSE distance := trajectory.P[i]-CSP_Config.MinimumPosition; END_IF
        CSP_Data.Axis[i].VelocityAllowed := MIN(CSP_Config.MaximumVelocity,
            SQRT(2.0*CSP_Config.BrakingAcceleration*MAX(0.0,distance)));
    END_FOR
70:
    // Reset handback: bring any active CSP command to rest in mode 8 first.
    CSP_Data.PlatformState := PlatformControlState.PP_HANDBACK;
    IF CSP_Data.Active THEN
        IF NOT allMode OR NOT allEnabled THEN
            CSP_Data.Fault := TRUE; CSP_Data.FaultCode := 6; RETURN;
        END_IF
        trajectory(Initialize:=FALSE, NewTarget:=FALSE, Stop:=TRUE);
        IF trajectory.Fault THEN CSP_Data.Fault := TRUE; CSP_Data.FaultCode := 7; RETURN; END_IF
        FOR i := 1 TO 6 DO
            CSP_Data.Axis[i].CommandPosition := trajectory.P[i];
            CSP_Data.Axis[i].CommandVelocity := trajectory.V[i];
            CSP_Data.Axis[i].CommandAcceleration := trajectory.A[i];
            CSP_Data.Axis[i].TargetRaw := LREAL_TO_DINT(trajectory.P[i]/CSP_Data.Axis[i].PositionFactor);
            CSP_Data.Axis[i].ModeRequested := 8;
            CSP_Data.Axis[i].Controlword := 16#000F;
        END_FOR
        IF NOT trajectory.Busy AND standstill.Q THEN
            FOR i := 1 TO 6 DO holdRaw[i] := CSP_Data.Axis[i].TargetRaw; END_FOR
            CSP_Data.Active := FALSE; CSP_Data.TransitionState := 71;
        END_IF
    ELSE
        // Handover hold or after quick stop: keep enabled axes at their current
        // CSP target; disabled/faulted axes get no enable and no fault reset.
        FOR i := 1 TO 6 DO
            IF CSP_Data.Axis[i].CiA402State = 16#0027 THEN
                holdRaw[i] := CSP_Data.Axis[i].TargetRaw;
            ELSE
                holdRaw[i] := CSP_Data.Axis[i].ActualRaw;
            END_IF
        END_FOR
        CSP_Data.TransitionState := 71;
    END_IF
71:
    // Request PP (mode 1) on all six drives while holding position. In PP mode a
    // target without a new-setpoint bit starts no motion.
    CSP_Data.PlatformState := PlatformControlState.PP_HANDBACK;
    FOR i := 1 TO 6 DO
        CSP_Data.Axis[i].TargetRaw := holdRaw[i];
        CSP_Data.Axis[i].ModeRequested := CSP_Config.CONTROL_MODE_PP;
        IF CSP_Data.Axis[i].CiA402State = 16#0027 THEN CSP_Data.Axis[i].Controlword := 16#000F;
        ELSE CSP_Data.Axis[i].Controlword := 16#0002; END_IF
    END_FOR
    // All six displays must confirm mode 1 (ModeBlockingAxis names a laggard);
    // otherwise the transition timeout raises FaultCode 1 with TimeoutState 71.
    IF allPPMode THEN
        // Mode 1 was already in the PDO image in earlier cycles. From this
        // cycle's CSP_WriteOutputs call the original Festo writer is the sole writer.
        CSP_Data.Active := FALSE; CSP_Data.ReadyToStart := FALSE;
        CSP_Data.ResetRequired := TRUE; CSP_Data.Homing := FALSE; homePhase := 0;
        CSP_Data.TransitionState := 0;
        CSP_Data.PlatformState := PlatformControlState.PP_RESET;
        resetRequest := FALSE;
        CSP_Data.CSPReleased := TRUE;
        CSP_Data.OwnsOutputs := FALSE;
    END_IF
END_CASE

END_PROGRAM

// PLC/Application/CSP_ReadAxis
FUNCTION CSP_ReadAxis : BOOL
VAR_INPUT
    Axis : REFERENCE TO AXIS_REF_CiA402_ETC_CMMT_AS;
    PlatformAxis : INT;
END_VAR

IF PlatformAxis < 1 OR PlatformAxis > 6 THEN RETURN; END_IF
CSP_Data.Axis[PlatformAxis].ReadinessCode := 1;

IF Axis.pIoStatusword = 0
    OR Axis.pIoModesOfOperationDisplay = 0
    OR Axis.pIoPositionActualValue = 0
    OR Axis.pIoVelocityActualValue = 0
    OR Axis.pIoControlword = 0
    OR Axis.pIoModesOfOperation = 0
    OR Axis.pIoTargetPosition = 0 THEN

    CSP_Data.Axis[PlatformAxis].Ready := FALSE;
    RETURN;
END_IF

CSP_Data.Axis[PlatformAxis].Statusword := Axis.pIoStatusword^;
CSP_Data.Axis[PlatformAxis].ModeActual := Axis.pIoModesOfOperationDisplay^;
CSP_Data.Axis[PlatformAxis].ActualRaw := Axis.pIoPositionActualValue^;
CSP_Data.Axis[PlatformAxis].ActualPosition := Axis.ActualPosition;
CSP_Data.Axis[PlatformAxis].ActualVelocity := Axis.ActualVelocity;

// Reuse Festo conversion factors.
CSP_Data.Axis[PlatformAxis].PositionFactor := Axis.rPositionFactor;
CSP_Data.Axis[PlatformAxis].VelocityFactor := Axis.rVelocityFactor;

CSP_Data.Axis[PlatformAxis].Ready :=
    Axis.SDOsInitialized
    AND Axis.rPositionFactor > 0
    AND (Axis.SlaveConnectorFlags AND 16#3F0) = 16#F0;

// Verify raw position conversion against Festo's calculated position.
IF Axis.rPositionFactor > 0 THEN

    CSP_Data.Axis[PlatformAxis].Ready :=
        CSP_Data.Axis[PlatformAxis].Ready
        AND ABS(
            DINT_TO_LREAL(Axis.pIoPositionActualValue^) * Axis.rPositionFactor
            - Axis.ActualPosition
        ) <= 0.01;

    CSP_Data.Axis[PlatformAxis].ActualPosition :=
        DINT_TO_LREAL(Axis.pIoPositionActualValue^) * Axis.rPositionFactor;

    CSP_Data.Axis[PlatformAxis].FollowingError :=
        DINT_TO_LREAL(CSP_Data.FollowingErrorRaw[PlatformAxis]) * Axis.rPositionFactor;

END_IF

CSP_Data.Axis[PlatformAxis].FollowingErrorRaw :=
    CSP_Data.FollowingErrorRaw[PlatformAxis];

// Keep the blocking condition visible even before TCP feedback is valid.
IF NOT Axis.SDOsInitialized THEN CSP_Data.Axis[PlatformAxis].ReadinessCode := 2;
ELSIF NOT (Axis.rPositionFactor > 0) THEN CSP_Data.Axis[PlatformAxis].ReadinessCode := 3;
ELSIF (Axis.SlaveConnectorFlags AND 16#3F0) <> 16#F0 THEN CSP_Data.Axis[PlatformAxis].ReadinessCode := 4;
ELSIF NOT CSP_Data.Axis[PlatformAxis].Ready THEN CSP_Data.Axis[PlatformAxis].ReadinessCode := 5;
ELSE CSP_Data.Axis[PlatformAxis].ReadinessCode := 0;
END_IF
CSP_ReadAxis := CSP_Data.Axis[PlatformAxis].Ready;

END_FUNCTION

// Axis
FUNCTION_BLOCK Axis
VAR
	// Power stage of the servo drive.
	MC_Power: MC_Power_Festo;
	// Reset object to reset servo drive.
	MC_Reset: MC_Reset_Festo;
	// Move absolute object to move the servo.
	MC_MoveAbsolute: MC_MoveAbsolute_Festo;
	// Read object to read current position.
	MC_ReadActualPosition: MC_ReadActualPosition_Festo;
	// Read status object to read current status of servo drive.
	MC_ReadStatus: MC_ReadStatus_Festo;
	
	// REF to axis.
	axis: REFERENCE TO AXIS_REF_FESTO;
	// Allow move orders to be overwritten by new moveorders.
	continuousUpdate: BOOL := FALSE;
	// Execute a move order.
	execute: BOOL := FALSE;
	// Drive is enabled.
	isEnabled: BOOL := FALSE;
	// Drive is in error.
	error: BOOL := FALSE;
	// Drive is beign reset, toggle bit.
	reset: BOOL := FALSE;
	// Requested position of servo.
	position: REAL := 0;
	// Requested velocity of servo.
	velocity: REAL := 0;
	// Acceleration of servo.
	acceleration: REAL := 5000;
	// Deceleration of servo.
	deceleration: REAL := 5000;
	// Jerk of servo.
	jerk: REAL := 15000;
END_VAR

PROPERTY enabled : BOOL
GET
enabled := THIS^.isEnabled AND (NOT THIS^.MC_ReadStatus.Disabled);
END_GET
SET
THIS^.isEnabled := enabled;
END_SET
END_PROPERTY

METHOD init : BOOL
VAR_INPUT
	axis : REFERENCE TO AXIS_REF_FESTO;
END_VAR
// This function references the servo drive to the instance of the function block.
THIS^.axis REF= axis;
END_METHOD

METHOD doAbort : BOOL
VAR_INPUT
END_VAR
THIS^.execute := FALSE;
END_METHOD

METHOD isReady : BOOL
VAR_INPUT
END_VAR
// Axis is ready when in standstill and not been given an execution order.
isReady := THIS^.MC_ReadStatus.Standstill AND NOT THIS^.execute;
END_METHOD

METHOD doMovement : BOOL
VAR_INPUT
	velocity: REAL := 0;
	position: REAL := 0;
	continuousUpdate: BOOL := FALSE;
END_VAR
// Only do movements when drive is started.
IF THIS^.isEnabled THEN
	THIS^.position := position;
	THIS^.velocity := velocity; 
	THIS^.continuousUpdate := continuousUpdate;
	THIS^.execute := TRUE;
	DoMovement := TRUE;		// return
ELSE
	THIS^.execute := FALSE;
	DoMovement := FALSE;	// return
END_IF;
END_METHOD

METHOD doReset
THIS^.reset := TRUE;
END_METHOD

METHOD getPosition : REAL
VAR_INPUT
END_VAR
IF THIS^.MC_ReadActualPosition.Valid OR (NOT THIS^.MC_ReadActualPosition.Error) THEN
	getPosition := THIS^.MC_ReadActualPosition.Position;
ELSE
	getPosition := -1;
END_IF
END_METHOD

METHOD inError : BOOL
VAR_INPUT
END_VAR
inError := THIS^.error;
END_METHOD

METHOD cycle : BOOL
VAR_INPUT
END_VAR
// Read drive status first
MC_ReadStatus(
	axis := THIS^.axis, 
	Enable := TRUE
);

// Set drive to error if an error occurs.
IF THIS^.MC_ReadStatus.ErrorStop OR THIS^.MC_ReadStatus.Error THEN
	THIS^.error := TRUE;
END_IF

// Function block to enable the drive.
THIS^.MC_Power(
	axis := THIS^.axis,
	Enable := THIS^.isEnabled
);

// Function block to reset the drive.
THIS^.MC_Reset(
	axis := THIS^.axis,
	Execute := THIS^.reset
);

// Reset the reset variable
IF (THIS^.MC_Reset.Done AND THIS^.reset) OR THIS^.MC_Reset.Error THEN
	THIS^.reset := FALSE;
	THIS^.error := FALSE;
END_IF

// Reset execute when movement is done.
IF (THIS^.MC_MoveAbsolute.Done AND NOT THIS^.continuousUpdate) OR THIS^.MC_MoveAbsolute.CommandAborted OR THIS^.error THEN
	THIS^.execute := FALSE;
END_IF

// Reset the move function if it's in error.
IF NOT THIS^.MC_MoveAbsolute.Error THEN
	// Function block to move the drive.
	THIS^.MC_MoveAbsolute(
		axis := THIS^.axis,
		Execute := THIS^.execute,
		ContinuousUpdate := THIS^.continuousUpdate,
		position := THIS^.position,
		velocity := THIS^.velocity,
		acceleration := THIS^.acceleration,
		deceleration := THIS^.deceleration,
		jerk := THIS^.jerk
	);
ELSE
	THIS^.MC_MoveAbsolute(axis := THIS^.axis, Execute := FALSE);
END_IF;

// Function block to read the drives current position.
THIS^.MC_ReadActualPosition(
	axis := THIS^.axis,
	Enable := TRUE
);
END_METHOD

METHOD isInitialised : BOOL
VAR_INPUT
END_VAR
isInitialised := THIS^.MC_ReadStatus.Valid;
END_METHOD

METHOD PPMoveDone : BOOL
// Level-based PP completion, as recorded by the original Axis.cycle():
// doMovement() sets execute, and cycle() clears it only after MC_MoveAbsolute
// Done (or CommandAborted/axis error). isReady() = drive Standstill AND NOT
// execute. The transient Done output itself is not used. The caller must also
// check the reached position, which excludes a move cleared by abort.
PPMoveDone := THIS^.isReady() AND NOT THIS^.error
    AND NOT THIS^.MC_MoveAbsolute.Error AND NOT THIS^.MC_MoveAbsolute.CommandAborted;
END_METHOD

END_FUNCTION_BLOCK

// PLC/Application/CSP_WriteOutputs
PROGRAM CSP_WriteOutputs

// Sole final writer, called after CSP_Cycle in the EtherCAT task.
CSP_WriteAxis(Axis:=servo_drive_1,PlatformAxis:=1);
CSP_WriteAxis(Axis:=servo_drive_2,PlatformAxis:=2);
CSP_WriteAxis(Axis:=servo_drive_3,PlatformAxis:=3);
CSP_WriteAxis(Axis:=servo_drive_4,PlatformAxis:=4);
CSP_WriteAxis(Axis:=servo_drive_5,PlatformAxis:=5);
CSP_WriteAxis(Axis:=servo_drive_6,PlatformAxis:=6);

END_PROGRAM

// PLC/Application/CSP_WriteAxis
FUNCTION CSP_WriteAxis : BOOL
VAR_INPUT
    Axis : REFERENCE TO AXIS_REF_CiA402_ETC_CMMT_AS;
    PlatformAxis : INT;
END_VAR

IF PlatformAxis < 1 OR PlatformAxis > 6 OR NOT CSP_Data.OwnsOutputs THEN
    Axis.BeforeWriteOutputs();
    IF PlatformAxis >= 1 AND PlatformAxis <= 6 AND Axis.pIoModesOfOperation <> 0
        AND Axis.pIoControlword <> 0 AND Axis.pIoTargetPosition <> 0 THEN
        CSP_Data.Axis[PlatformAxis].ModeRequested := Axis.pIoModesOfOperation^;
        CSP_Data.Axis[PlatformAxis].Controlword := Axis.pIoControlword^;
        CSP_Data.Axis[PlatformAxis].TargetRaw := Axis.pIoTargetPosition^;
    END_IF
ELSE
    // These are the SAME PDO pointers initialized by the existing Festo device.
    // Do not run its PP writer and then race it from another IEC task.
    IF Axis.pIoControlword <> 0 AND Axis.pIoModesOfOperation <> 0 AND Axis.pIoTargetPosition <> 0 THEN
        Axis.pIoTargetPosition^ := CSP_Data.Axis[PlatformAxis].TargetRaw;
        Axis.pIoModesOfOperation^ := CSP_Data.Axis[PlatformAxis].ModeRequested;
        Axis.pIoControlword^ := CSP_Data.Axis[PlatformAxis].Controlword;
        IF Axis.pIoVelocityOffset <> 0 THEN Axis.pIoVelocityOffset^ := 0; END_IF
        IF Axis.pIoTorqueOffset <> 0 THEN Axis.pIoTorqueOffset^ := 0; END_IF
    END_IF
END_IF

END_FUNCTION

// PLC/Application/CSP_Trajectory6
FUNCTION_BLOCK CSP_Trajectory6
VAR_INPUT
    Initialize, NewTarget, Stop : BOOL;
    Actual, Requested : ARRAY[1..6] OF LREAL;
END_VAR
VAR_OUTPUT
    P, V, A : ARRAY[1..6] OF LREAL;
    // Busy: not yet at rest on the latest target. Braking: Stop in progress.
    // Deferred: some axis passes its target before reversing (unavoidable with
    // the current V/A and the acceleration/jerk limits).
    Busy, Braking, Deferred, Fault : BOOL;
END_VAR
VAR CONSTANT
    MaximumRampSeconds : LREAL := 0.1; // >= PC send period (nominal 50 ms)
    Iterations : INT := 20; // bisection steps: 2*MaximumJerk / 2^20 resolution
END_VAR
VAR
    goal, rampStart, rampEnd : ARRAY[1..6] OF LREAL;
    rampElapsed, rampDuration, sinceTarget : LREAL;
    stopping : BOOL;
    cycleTime, maxV, maxA, maxJ : LREAL;
    jHigh, jLow, jTry, lo, hi, p1, v1, a1, rest : LREAL;
    i, k : INT;
    ok : BOOL;
END_VAR

// Online, receding-horizon generator. Every CSP cycle each axis independently
// chooses one jerk value from its CURRENT commanded P/V/A, so P, V and A are
// always continuous and a new target simply changes the next choice; there is
// no stop-at-target plan to finish and no separate brake-to-standstill path.
// The chosen jerk is the one whose resulting state, braked at full limits,
// comes to rest closest to the target (a time-optimal approach). It is limited
// by MaximumJerk, MaximumAcceleration/BrakingAcceleration, a jerk-aware
// MaximumVelocity envelope, and a travel envelope: from every commanded state
// a full-limit stop ends inside MinimumPosition..MaximumPosition.
// The 20 Hz targets are linearly interpolated over the measured packet
// interval, starting from the current interpolated target (one packet delay).
cycleTime := CSP_Config.CycleSeconds;
maxV := CSP_Config.MaximumVelocity;
maxA := MIN(CSP_Config.MaximumAcceleration, CSP_Config.BrakingAcceleration);
maxJ := CSP_Config.MaximumJerk;
IF Initialize THEN
    P := Actual; goal := Actual; rampStart := Actual; rampEnd := Actual;
    FOR i := 1 TO 6 DO V[i] := 0; A[i] := 0; END_FOR
    rampDuration := MAX(cycleTime, 1E-3); rampElapsed := rampDuration;
    sinceTarget := MaximumRampSeconds; stopping := FALSE;
    Busy := FALSE; Braking := FALSE; Deferred := FALSE;
    Fault := cycleTime <= 0 OR maxV <= 0 OR maxA <= 0 OR maxJ <= 0
        OR CSP_Config.MinimumPosition >= CSP_Config.MaximumPosition;
    RETURN;
END_IF
IF Fault THEN RETURN; END_IF

IF Stop THEN
    IF NOT stopping THEN
        // Target = where a full-limit stop from the current state ends.
        FOR i := 1 TO 6 DO
            goal[i] := P[i] + CSP_StopOffset(V:=V[i], A:=A[i], MaxAcceleration:=maxA, MaxJerk:=maxJ);
        END_FOR
        rampStart := goal; rampEnd := goal; rampElapsed := rampDuration;
        stopping := TRUE;
    END_IF
ELSE
    stopping := FALSE;
    IF NewTarget THEN
        // Retarget immediately from the current interpolated target: no jump.
        FOR i := 1 TO 6 DO
            rampStart[i] := goal[i];
            rampEnd[i] := LIMIT(CSP_Config.MinimumPosition, Requested[i], CSP_Config.MaximumPosition);
        END_FOR
        rampDuration := LIMIT(2.0*cycleTime, sinceTarget, MaximumRampSeconds);
        rampElapsed := 0; sinceTarget := 0;
    END_IF
END_IF
sinceTarget := MIN(sinceTarget + cycleTime, MaximumRampSeconds);
rampElapsed := MIN(rampDuration, rampElapsed + cycleTime);

Busy := FALSE; Deferred := FALSE;
FOR i := 1 TO 6 DO
    IF rampElapsed >= rampDuration THEN
        goal[i] := rampEnd[i]; // exact: lets Busy clear at rest
    ELSE
        goal[i] := rampStart[i] + (rampEnd[i] - rampStart[i])*rampElapsed/rampDuration;
    END_IF
    IF rampElapsed >= rampDuration AND ABS(A[i]) <= maxJ*cycleTime AND ABS(V[i]) <= maxJ*cycleTime*cycleTime
        AND ABS(P[i] - goal[i]) <= maxJ*cycleTime*cycleTime*cycleTime THEN
        // Terminal capture: the remaining stop is shorter than one cycle. The
        // change is within one cycle of full jerk; it prevents a +/- limit cycle.
        P[i] := goal[i]; V[i] := 0; A[i] := 0;
    ELSE
        jHigh := MIN(maxJ, (maxA - A[i])/cycleTime);
        jLow := MAX(-maxJ, (-maxA - A[i])/cycleTime);
        // Upper envelope: velocity peak after unwinding A, and stop below MaximumPosition.
        jTry := jHigh;
        p1 := P[i] + V[i]*cycleTime + A[i]*cycleTime*cycleTime/2.0 + jTry*cycleTime*cycleTime*cycleTime/6.0;
        v1 := V[i] + A[i]*cycleTime + jTry*cycleTime*cycleTime/2.0;
        a1 := A[i] + jTry*cycleTime;
        ok := v1 + MAX(a1, 0.0)*MAX(a1, 0.0)/(2.0*maxJ) <= maxV
            AND p1 + CSP_StopOffset(V:=v1, A:=a1, MaxAcceleration:=maxA, MaxJerk:=maxJ)
            <= CSP_Config.MaximumPosition;
        IF NOT ok THEN
            lo := jLow; hi := jHigh;
            FOR k := 1 TO Iterations DO
                jTry := (lo + hi)/2.0;
                p1 := P[i] + V[i]*cycleTime + A[i]*cycleTime*cycleTime/2.0 + jTry*cycleTime*cycleTime*cycleTime/6.0;
                v1 := V[i] + A[i]*cycleTime + jTry*cycleTime*cycleTime/2.0;
                a1 := A[i] + jTry*cycleTime;
                ok := v1 + MAX(a1, 0.0)*MAX(a1, 0.0)/(2.0*maxJ) <= maxV
                    AND p1 + CSP_StopOffset(V:=v1, A:=a1, MaxAcceleration:=maxA, MaxJerk:=maxJ)
                        <= CSP_Config.MaximumPosition;
                IF ok THEN lo := jTry; ELSE hi := jTry; END_IF
            END_FOR
            jHigh := lo;
        END_IF
        // Lower envelope: velocity trough and stop above MinimumPosition.
        jTry := jLow;
        p1 := P[i] + V[i]*cycleTime + A[i]*cycleTime*cycleTime/2.0 + jTry*cycleTime*cycleTime*cycleTime/6.0;
        v1 := V[i] + A[i]*cycleTime + jTry*cycleTime*cycleTime/2.0;
        a1 := A[i] + jTry*cycleTime;
        ok := v1 - MIN(a1, 0.0)*MIN(a1, 0.0)/(2.0*maxJ) >= -maxV
            AND p1 + CSP_StopOffset(V:=v1, A:=a1, MaxAcceleration:=maxA, MaxJerk:=maxJ)
            >= CSP_Config.MinimumPosition;
        IF NOT ok THEN
            lo := jLow; hi := jHigh;
            FOR k := 1 TO Iterations DO
                jTry := (lo + hi)/2.0;
                p1 := P[i] + V[i]*cycleTime + A[i]*cycleTime*cycleTime/2.0 + jTry*cycleTime*cycleTime*cycleTime/6.0;
                v1 := V[i] + A[i]*cycleTime + jTry*cycleTime*cycleTime/2.0;
                a1 := A[i] + jTry*cycleTime;
                ok := v1 - MIN(a1, 0.0)*MIN(a1, 0.0)/(2.0*maxJ) >= -maxV
                    AND p1 + CSP_StopOffset(V:=v1, A:=a1, MaxAcceleration:=maxA, MaxJerk:=maxJ)
                        >= CSP_Config.MinimumPosition;
                IF ok THEN hi := jTry; ELSE lo := jTry; END_IF
            END_FOR
            jLow := hi;
        END_IF
        IF jLow > jHigh THEN
            // Not reachable from a state this block produced; reduce |A| only.
            jTry := LIMIT(-maxJ, -A[i]/cycleTime, maxJ);
        ELSE
            // Rest point after this cycle rises monotonically with jerk: choose
            // the jerk whose rest point is the target, clamped to the envelope.
            jTry := jHigh;
            p1 := P[i] + V[i]*cycleTime + A[i]*cycleTime*cycleTime/2.0 + jTry*cycleTime*cycleTime*cycleTime/6.0;
            v1 := V[i] + A[i]*cycleTime + jTry*cycleTime*cycleTime/2.0;
            a1 := A[i] + jTry*cycleTime;
            rest := p1 + CSP_StopOffset(V:=v1, A:=a1, MaxAcceleration:=maxA, MaxJerk:=maxJ);
            IF rest > goal[i] THEN
                jTry := jLow;
                p1 := P[i] + V[i]*cycleTime + A[i]*cycleTime*cycleTime/2.0 + jTry*cycleTime*cycleTime*cycleTime/6.0;
                v1 := V[i] + A[i]*cycleTime + jTry*cycleTime*cycleTime/2.0;
                a1 := A[i] + jTry*cycleTime;
                rest := p1 + CSP_StopOffset(V:=v1, A:=a1, MaxAcceleration:=maxA, MaxJerk:=maxJ);
                IF rest < goal[i] THEN
                    lo := jLow; hi := jHigh;
                    FOR k := 1 TO Iterations DO
                        jTry := (lo + hi)/2.0;
                        p1 := P[i] + V[i]*cycleTime + A[i]*cycleTime*cycleTime/2.0 + jTry*cycleTime*cycleTime*cycleTime/6.0;
                        v1 := V[i] + A[i]*cycleTime + jTry*cycleTime*cycleTime/2.0;
                        a1 := A[i] + jTry*cycleTime;
                        rest := p1 + CSP_StopOffset(V:=v1, A:=a1, MaxAcceleration:=maxA, MaxJerk:=maxJ);
                        IF rest > goal[i] THEN hi := jTry; ELSE lo := jTry; END_IF
                    END_FOR
                    jTry := lo;
                END_IF
            END_IF
        END_IF
        // Exact cubic integration over one cycle.
        P[i] := P[i] + V[i]*cycleTime + A[i]*cycleTime*cycleTime/2.0 + jTry*cycleTime*cycleTime*cycleTime/6.0;
        V[i] := V[i] + A[i]*cycleTime + jTry*cycleTime*cycleTime/2.0;
        A[i] := A[i] + jTry*cycleTime;
    END_IF
    IF P[i] < CSP_Config.MinimumPosition - 1E-6 OR P[i] > CSP_Config.MaximumPosition + 1E-6 THEN
        Fault := TRUE;
    END_IF
    rest := P[i] + CSP_StopOffset(V:=V[i], A:=A[i], MaxAcceleration:=maxA, MaxJerk:=maxJ);
    Deferred := Deferred OR (V[i]*(goal[i] - rest) < 0 AND ABS(goal[i] - rest) > 1E-3);
    Busy := Busy OR V[i] <> 0 OR A[i] <> 0 OR P[i] <> rampEnd[i];
END_FOR
Braking := stopping AND Busy;

END_FUNCTION_BLOCK

// PLC/Application/CSP_StopOffset
FUNCTION CSP_StopOffset : LREAL
VAR_INPUT
    V, A : LREAL;
    MaxAcceleration, MaxJerk : LREAL;
END_VAR
VAR
    t : ARRAY[1..3] OF LREAL;
    sign, speed, accel, peak, h, jk, sp, sv, sa : LREAL;
    k : INT;
END_VAR

// Signed displacement of the minimum-time jerk-limited stop (V = A = 0) from
// (V, A): jerk -J, optional constant -peak, jerk +J (mirrored by sign). The braking
// direction is the sign of the velocity left after unwinding A at full jerk, so
// every state is valid, including one that must cross zero velocity first.
// The result increases monotonically with V and A.
CSP_StopOffset := 0;
IF MaxJerk <= 0 OR MaxAcceleration <= 0 THEN RETURN; END_IF
sign := 1.0;
IF V + A*ABS(A)/(2.0*MaxJerk) < 0 THEN sign := -1.0; END_IF
speed := sign*V; accel := sign*A;
IF ABS(speed) < 1E-12 AND ABS(accel) < 1E-12 THEN RETURN; END_IF
peak := MIN(MaxAcceleration, SQRT(MAX(0.0, MaxJerk*speed + accel*accel/2.0)));
t[1] := MAX(0.0, (accel + peak)/MaxJerk);
t[2] := 0;
IF peak > 0 THEN
    t[2] := MAX(0.0, (speed + (accel*accel - 2.0*peak*peak)/(2.0*MaxJerk))/peak);
END_IF
t[3] := peak/MaxJerk;
sp := 0; sv := speed; sa := accel;
FOR k := 1 TO 3 DO
    CASE k OF
        1: jk := -MaxJerk;
        2: jk := 0;
    ELSE
        jk := MaxJerk;
    END_CASE
    h := t[k];
    sp := sp + sv*h + sa*h*h/2.0 + jk*h*h*h/6.0;
    sv := sv + sa*h + jk*h*h/2.0;
    sa := sa + jk*h;
END_FOR
CSP_StopOffset := sign*sp;

END_FUNCTION

// PLC/Application/main
PROGRAM main
VAR
	bInit: BOOL := TRUE;
	iCounter : INT;
	bEnabled: BOOL;
	iDataUpdated: INT := 0;
	tonTimer: TON;
	UpdateCount: INT := 0;
    cspStartEdge : R_TRIG;
END_VAR

cspStartEdge(CLK:=GVL.startButton OR GVL.startHMI);
// ============================================================================
// COMMON OPERATOR CONTROL
// This section runs in BOTH PP and CSP mode.
// ============================================================================

// Safety/E-stop has highest priority.
// Also clear bEnabled so releasing the E-stop cannot automatically restart.
IF NOT GVL.safetySystem THEN
    bEnabled := FALSE;

// Reset stops the system and requires a new Start afterwards.
ELSIF GVL.resetButton OR GVL.resetHMI THEN
    bEnabled := FALSE;

// Stop buttons.
ELSIF GVL.stopButton OR GVL.stopHMI THEN
    bEnabled := FALSE;

// Start is only accepted while the safety system is OK.
ELSIF (GVL.startButton OR GVL.startHMI)
    AND (CSP_Config.ControlMode <> CSP_Config.CONTROL_MODE_CSP OR cspStartEdge.Q) THEN
    bEnabled := TRUE;
END_IF;


// ============================================================================
// CSP MODE
// ============================================================================
IF CSP_Config.ControlMode = CSP_Config.CONTROL_MODE_CSP THEN
    // Policy 8 uses the working PP reset/start, then automatic CSP ownership.
    PlatformStartup();

ELSE

    // CSP must not retain control while PP is selected.
    CSP_Data.Enable := FALSE;
    CSP_Data.Reset := FALSE;


    // ------------------------------------------------------------------------
    // Existing PP initialization.
    // ------------------------------------------------------------------------
    IF bInit THEN

        GVL.FlightSimulator.init(
            axis1 := servo_drive_1,
            axis2 := servo_drive_2,
            axis3 := servo_drive_3,
            axis4 := servo_drive_4,
            axis5 := servo_drive_5,
            axis6 := servo_drive_6,
            GVL.lightRed,
            GVL.lightYellow,
            GVL.lightGreen,
            enabled := bEnabled,
            safetySystem := GVL.safetySystem,
            newPositions := GVL.servoPositions,
            newVelocities := GVL.servoVelocities
        );

        bInit := FALSE;

    END_IF


    // ------------------------------------------------------------------------
    // Existing PP reset behavior.
    // ------------------------------------------------------------------------
    IF GVL.resetButton OR GVL.resetHMI THEN

        GVL.FlightSimulator.doReset();

        // Reset PP position data so the platform does not move toward an
        // old position after resetting.
        FOR iCounter := 1 TO 6 DO

            GVL.currentPositions[iCounter].Number := 0.0;
            GVL.servoPositions[iCounter] := 0.0;
            GVL.servoVelocities[iCounter] := 0.0;

        END_FOR

    END_IF


    // ------------------------------------------------------------------------
    // Existing PP command-data handling.
    // ------------------------------------------------------------------------
    FOR iCounter := 1 TO 6 BY 1 DO

        IF GVL.useTCPData THEN

            // Use latest TCP data.
            GVL.servoPositions[iCounter] :=
                tcpClient.servoData.positions[iCounter].Number;

            GVL.servoVelocities[iCounter] :=
                tcpClient.servoData.speeds[iCounter].Number;

            // Diagnostic counter.
            IF tcpClient.parseJSON.Done THEN
                UpdateCount := UpdateCount + 1;
            END_IF

        ELSE

            // Manual HMI control.
            GVL.servoPositions[iCounter] :=
                GVL.nextPositionInput;

            GVL.servoVelocities[iCounter] :=
                GVL.nextVelocityInput;

        END_IF

    END_FOR


    // ------------------------------------------------------------------------
    // Run the ORIGINAL PP motion controller.
    //
    // IMPORTANT:
    // This must NEVER execute in CSP mode because it would cause the old
    // Festo PP controller and the new CSP controller to compete for the drives.
    // ------------------------------------------------------------------------
    GVL.FlightSimulator.cycle();


    // ------------------------------------------------------------------------
    // Existing PP actual-position feedback.
    // ------------------------------------------------------------------------
    FOR iCounter := 1 TO 6 BY 1 DO

        GVL.currentPositions[iCounter].Number :=
            GVL.FlightSimulator.axis[iCounter].getPosition();

        GVL.servoPositionsCurrent[iCounter] :=
            GVL.FlightSimulator.axis[iCounter].getPosition();

    END_FOR

END_IF

END_PROGRAM

// PLC/Application/PlatformStartup
PROGRAM PlatformStartup
VAR
    initialized : BOOL;
    ppEnabled : BOOL;
    resetButtonEdge, startButtonEdge : R_TRIG;
    ppStartArmed : BOOL;
    ppState : stateFlightSimulator;
    allPPMode, allInTravel, allAtNeutral : BOOL;
    atNeutral : ARRAY[1..6] OF BOOL;
    i : INT;
END_VAR

// Called only for the PP-startup/CSP-runtime policy. Pure PP main is unchanged.
// Ownership: PP (this task) until PPReleased; CSP (EtherCAT task) while
// CSP_Data.OwnsOutputs; PP again after CSP publishes CSPReleased on Reset.
resetButtonEdge(CLK:=GVL.resetButton OR GVL.resetHMI);
startButtonEdge(CLK:=GVL.startButton OR GVL.startHMI);
CSP_Data.Reset := GVL.resetButton OR GVL.resetHMI;
CSP_Data.StopRequested := GVL.stopButton OR GVL.stopHMI;

IF NOT initialized THEN
    GVL.FlightSimulator.init(
        axis1:=servo_drive_1, axis2:=servo_drive_2, axis3:=servo_drive_3,
        axis4:=servo_drive_4, axis5:=servo_drive_5, axis6:=servo_drive_6,
        lightRed:=GVL.lightRed, lightYellow:=GVL.lightYellow, lightGreen:=GVL.lightGreen,
        enabled:=ppEnabled, safetySystem:=GVL.safetySystem,
        newPositions:=GVL.servoPositions, newVelocities:=GVL.servoVelocities);
    initialized := TRUE;
END_IF

// Reset handback: CSP braked, restored mode 1 on all six drives and no longer
// writes them. Take ownership back and run the ORIGINAL PP reset from here.
IF CSP_Data.PPReleased AND CSP_Data.CSPReleased THEN
    CSP_Data.PPReleased := FALSE;
    ppEnabled := FALSE; ppStartArmed := FALSE;
    FOR i := 1 TO 6 DO CSP_Data.PPMoveDone[i] := FALSE; END_FOR
    // Without safety, FlightSimulator.cycle() immediately selects its error state.
    GVL.FlightSimulator.doReset();
END_IF

// PPReleased is published AFTER the final complete PP call. Once published,
// this task NEVER calls a PP motion block again until CSPReleased. Only the CSP
// task changes OwnsOutputs, at its cycle boundary, after capturing all six
// actual positions.
IF CSP_Data.PPReleased THEN
    IF NOT GVL.safetySystem OR CSP_Data.StopRequested OR CSP_Data.Reset OR CSP_Data.Fault THEN
        ppEnabled := FALSE;
    ELSIF startButtonEdge.Q AND CSP_Data.ReadyToStart THEN
        ppEnabled := TRUE;
    END_IF
    CSP_Data.Enable := ppEnabled AND GVL.safetySystem;
    GVL.lightRed := NOT GVL.safetySystem OR CSP_Data.Fault;
    GVL.lightGreen := NOT GVL.lightRed AND CSP_Data.Active AND CSP_Data.ReadyToStart;
    GVL.lightYellow := NOT GVL.lightRed AND NOT GVL.lightGreen;
    FOR i := 1 TO 6 DO
        GVL.currentPositions[i].Number := LREAL_TO_REAL(CSP_Data.Axis[i].ActualPosition);
        GVL.servoPositionsCurrent[i] := LREAL_TO_REAL(CSP_Data.Axis[i].ActualPosition);
        GVL.servoPositions[i] := LREAL_TO_REAL(CSP_Data.Axis[i].RequestedPosition);
        GVL.servoVelocities[i] := LREAL_TO_REAL(CSP_Data.Axis[i].CommandVelocity);
    END_FOR
    RETURN;
END_IF

// Original PP reset on the button edge. The request is not stored: a Reset
// pressed during an E-stop cannot cause motion when the E-stop is released.
IF resetButtonEdge.Q THEN
    ppEnabled := FALSE; ppStartArmed := FALSE;
    FOR i := 1 TO 6 DO CSP_Data.PPMoveDone[i] := FALSE; END_FOR
    GVL.FlightSimulator.doReset();
END_IF
ppState := GVL.FlightSimulator.PPState();
IF NOT GVL.safetySystem OR CSP_Data.StopRequested THEN
    ppEnabled := FALSE;
ELSIF startButtonEdge.Q AND ppState = stateFlightSimulator.stopped AND NOT CSP_Data.CSPReleased THEN
    ppEnabled := TRUE; ppStartArmed := TRUE;
    FOR i := 1 TO 6 DO CSP_Data.PPMoveDone[i] := FALSE; END_FOR
END_IF
// Never feed PC targets to PP during startup. The original startup method
// selects position 200 and velocity 25 itself; these arrays are only a hold.
FOR i := 1 TO 6 DO GVL.servoPositions[i] := 200; GVL.servoVelocities[i] := 25; END_FOR
GVL.FlightSimulator.cycle(StartupOnly:=TRUE);
ppState := GVL.FlightSimulator.PPState();
CSP_Data.AllPPMoveDone := TRUE;
allPPMode := TRUE; allInTravel := TRUE; allAtNeutral := TRUE;
FOR i := 1 TO 6 DO
    // Evaluated every cycle from PP's own durable state; nothing is latched.
    // STARTED is entered one cycle after goNeutralPosition() sets execute, so
    // a ready axis in STARTED has finished that neutral move (or was aborted;
    // the position check below rejects that case).
    atNeutral[i] := ABS(CSP_Data.Axis[i].ActualPosition - CSP_Config.HomePosition)
        <= CSP_Config.HomeTolerance;
    allAtNeutral := allAtNeutral AND atNeutral[i];
    CSP_Data.PPMoveDone[i] := ppStartArmed AND ppState = stateFlightSimulator.started
        AND GVL.FlightSimulator.axis[i].PPMoveDone() AND atNeutral[i];
    CSP_Data.AllPPMoveDone := CSP_Data.AllPPMoveDone AND CSP_Data.PPMoveDone[i];
    allPPMode := allPPMode AND CSP_Data.Axis[i].ModeActual = CSP_Config.CONTROL_MODE_PP;
    allInTravel := allInTravel AND CSP_Data.Axis[i].ActualPosition >= CSP_Config.MinimumPosition
        AND CSP_Data.Axis[i].ActualPosition <= CSP_Config.MaximumPosition;
    GVL.currentPositions[i].Number := GVL.FlightSimulator.axis[i].getPosition();
    GVL.servoPositionsCurrent[i] := GVL.currentPositions[i].Number;
END_FOR
CSP_Data.Fault := ppState = stateFlightSimulator.error OR GVL.FlightSimulator.inError();
CSP_Data.FaultCode := 0;
IF CSP_Data.Fault THEN CSP_Data.FaultCode := 9; END_IF // inspect original PP/axis error
CSP_Data.Homing := FALSE;
CSP_Data.ReadyToStart := FALSE;
CSP_Data.Enable := ppEnabled AND GVL.safetySystem;
CASE ppState OF
    stateFlightSimulator.error:
        CSP_Data.PlatformState := PlatformControlState.FAULT;
        CSP_Data.ResetRequired := TRUE; ppEnabled := FALSE;
    stateFlightSimulator.resetting:
        CSP_Data.PlatformState := PlatformControlState.PP_RESET;
        CSP_Data.ResetRequired := TRUE;
    stateFlightSimulator.stopped:
        CSP_Data.PlatformState := PlatformControlState.PP_STOPPED;
        CSP_Data.ResetRequired := FALSE;
ELSE
    CSP_Data.PlatformState := PlatformControlState.PP_STARTING;
END_CASE
// PP startup finished: Start accepted, PP in STARTED, every axis ready with its
// neutral move complete (PPMoveDone) and within HomeTolerance of HomePosition
// (= goNeutralPosition's 200), and measured standstill for 200 ms.
CSP_Data.PPStartupComplete := ppStartArmed AND ppEnabled AND GVL.safetySystem
    AND NOT CSP_Data.Fault AND ppState = stateFlightSimulator.started
    AND GVL.FlightSimulator.isReady() AND CSP_Data.AllPPMoveDone AND CSP_Data.AllStationary;
IF CSP_Data.Fault THEN CSP_Data.StartupBlockReason := 7;
ELSIF NOT GVL.safetySystem THEN CSP_Data.StartupBlockReason := 3;
ELSIF NOT ppEnabled OR NOT ppStartArmed THEN CSP_Data.StartupBlockReason := 4;
ELSIF ppState <> stateFlightSimulator.started THEN CSP_Data.StartupBlockReason := 10;
ELSIF NOT GVL.FlightSimulator.isReady() THEN CSP_Data.StartupBlockReason := 12;
ELSIF NOT allAtNeutral THEN CSP_Data.StartupBlockReason := 13;
ELSIF NOT CSP_Data.AllPPMoveDone THEN CSP_Data.StartupBlockReason := 14;
ELSIF NOT CSP_Data.AllStationary THEN CSP_Data.StartupBlockReason := 11;
ELSIF NOT CSP_Config.Commissioned THEN CSP_Data.StartupBlockReason := 1;
ELSIF NOT allPPMode THEN CSP_Data.StartupBlockReason := 6;
ELSIF NOT allInTravel THEN CSP_Data.StartupBlockReason := 2;
ELSE CSP_Data.StartupBlockReason := 0;
END_IF
// The CSP task repeats these checks race-free when it captures the positions.
IF CSP_Data.PPStartupComplete AND CSP_Config.Commissioned AND allPPMode AND allInTravel
    AND NOT CSP_Data.CSPReleased THEN
    CSP_Data.PlatformState := PlatformControlState.CSP_HANDOVER;
    // Last write: cannot be observed until all PP motion calls above finished.
    CSP_Data.PPReleased := TRUE;
END_IF

END_PROGRAM

// FlightSimulator
FUNCTION_BLOCK FlightSimulator
VAR_OUTPUT
	// Axis objects.
	axis: ARRAY[1..6] OF Axis;
	// Signal objects.
	signal: signal;
END_VAR
VAR
	// Current state of flight simulator.
	state: stateFlightSimulator;
	// Used in some states to add extra delay.
	bToggle: BOOL;
	// REF to if system should be enabled.
	enabled: REFERENCE TO BOOL;
	// REF to safety system.
	safetySystem: REFERENCE TO BOOL;
	// REF to new positions.
	newPositions: REFERENCE TO ARRAY[1..6] OF REAL;
	// REF to new velocities.
	newVelocities: REFERENCE TO ARRAY[1..6] OF REAL;
END_VAR

METHOD safetyStop : BOOL
VAR
	// Counter to cycle through axis.
	iCounter: UINT;
END_VAR
// Disable all axis.
FOR iCounter := 1 TO 6 BY 1 DO
	THIS^.axis[iCounter].enabled := FALSE;
END_FOR
THIS^.enabled := FALSE;
END_METHOD

METHOD doReset : BOOL
VAR_INPUT
END_VAR
VAR
	// Counter to cycle through axis.
	iCounter: UINT;
END_VAR
THIS^.state := stateFlightSimulator.resetting;
END_METHOD

METHOD isEnabled : BOOL;
VAR_INPUT
END_VAR
VAR
	// Counter to cycle through axis.
	iCounter: INT;
END_VAR
// Check enabled status of all axis, when one is not enabled return with FALSE.
FOR iCounter := 1 TO 6 BY 1 DO
	IF NOT THIS^.axis[iCounter].enabled THEN
		isEnabled := FALSE;
		RETURN;
	END_IF;
END_FOR;

isEnabled := TRUE;
END_METHOD

METHOD getPositions : ARRAY[1..6] OF REAL
VAR_INPUT
END_VAR
VAR
	// Counter to cycle through axis.
	iCounter: INT;
END_VAR
// Write current axis positions
FOR iCounter := 1 TO 6 BY 1 DO
	getPositions[iCounter] := THIS^.axis[iCounter].getPosition();
END_FOR
END_METHOD

METHOD cycle : BOOL
VAR_INPUT
    StartupOnly : BOOL := FALSE; // PP startup for automatic CSP handover
END_VAR
VAR
	// Counter to cycle through axis.
	iCounter: UINT;
END_VAR
// If safety system has been triggered/broken go to error.
IF NOT THIS^.safetySystem THEN
	THIS^.state := stateFlightSimulator.error;
	THIS^.safetyStop();
END_IF

// If any Axis is in error stop all axis.
IF THIS^.inError() AND NOT (THIS^.state = stateFlightSimulator.error) THEN
	IF NOT (THIS^.state = stateFlightSimulator.resetting) THEN
		THIS^.state := stateFlightSimulator.error;
		THIS^.safetyStop();
	END_IF
END_IF

// Reset signal variables.
THIS^.signal.red.enable := FALSE;
THIS^.signal.yellow.enable := FALSE;
THIS^.signal.green.enable := FALSE;
THIS^.signal.red.blink := FALSE;
THIS^.signal.yellow.blink := FALSE;
THIS^.signal.green.blink := FALSE;

// Status case switch.
CASE THIS^.state OF
	stateFlightSimulator.stopped:
		// In STOPPED state:
		// Signal needs to be continuously yellow.
		// Drives needs to be disabled.
		// When enabled go to STARTING state.
		
		// Set signal.
		THIS^.signal.yellow.enable := TRUE;
		
		// Disable drives.
		IF THIS^.isEnabled() THEN
			FOR iCounter := 1 TO 6 BY 1 DO
				Axis[iCounter].enabled := FALSE;
			END_FOR
		END_IF
		
		// If flightsim is enabled go to STARTING state.
		IF THIS^.enabled THEN
			THIS^.state := stateFlightSimulator.starting;
		END_IF
		
	stateFlightSimulator.starting:
		// In STARTING state:
		// Signal needs to be blinking green.
		// Drives needs to be enabled.
		// Once enabled go to neutral position.
		// Once in neutral position go to STARTED state.
	
		// Set signal.
		THIS^.signal.green.enable := TRUE;
		THIS^.signal.green.blink := TRUE;
		
		// Start Axises.
		IF NOT THIS^.isEnabled() THEN
			FOR iCounter := 1 TO 6 BY 1 DO
				Axis[iCounter].enabled := TRUE;
				GVL.servoPositions[iCounter] := 200;
			END_FOR
		END_IF
		
		IF THIS^.isEnabled() AND THIS^.isReady() THEN
			IF NOT bToggle THEN
				// Move pistons to neutral position.
				THIS^.goNeutralPosition();
				bToggle := TRUE;
			ELSE
				// When position has been reached go to started state.
				bToggle := FALSE;
				THIS^.state := stateFlightSimulator.started;
			END_IF	
		END_IF
		
	stateFlightSimulator.started:
		// In STARTED state:
		// Signal needs to be continuously green.
		// When at least one of the drives goes to disabled go to ERROR state.
		// Do movement.
		// When not enabled go to STOPPING state.
	
		// Set signal.
		THIS^.signal.green.enable := TRUE;
		
		// If drives are disabled somehow go to error.
		IF NOT THIS^.isEnabled() THEN
			THIS^.state := stateFlightSimulator.error;
		END_IF
		
		// Do movement.
		// PP startup holds its completed neutral move until the CSP task takes over.
        IF NOT StartupOnly THEN
            THIS^.doMovement(THIS^.newPositions, THIS^.newVelocities);
        END_IF
		
		// If flightsim is disabled go to STOPPING state.
		IF NOT THIS^.enabled THEN
			THIS^.state := stateFlightSimulator.stopping;
		END_IF
		
	stateFlightSimulator.stopping:
		// In STOPPING state:
		// Signal needs to be blinking green.
		// Drives needs to be enabled.
		// Once enabled go to home position.
		// Once in home position go to STOPPED state.
	
		// Set signal.
		THIS^.signal.green.enable := TRUE;
		THIS^.signal.green.blink := TRUE;
		
		// Enable drives if not enabled yet.
		IF NOT THIS^.isEnabled() THEN
			FOR iCounter := 1 TO 6 BY 1 DO
				Axis[iCounter].enabled := TRUE;
			END_FOR
		END_IF
		
		IF THIS^.isEnabled() THEN
			IF NOT bToggle THEN
				// Move pistons to home position.
				THIS^.goHomePosition();
				bToggle := TRUE;
			ELSE
				IF THIS^.isReady() THEN
					// When position has been reached go to stopped state.
					bToggle := FALSE;
					THIS^.state := stateFlightSimulator.stopped;
				END_IF
			END_IF
		END_IF
		
	stateFlightSimulator.error:
		// In ERROR state:
		// Signal needs to be blinking red.
		
		// Set signal.
		THIS^.signal.red.enable := TRUE;
		THIS^.signal.red.blink := TRUE;
		
	stateFlightSimulator.resetting:
		// In RESETTING state:
		// Signal needs to be blinking yellow.
		// If in error drives needs to be reset.
		// Else go to home and go to STOPPED state.
	
		// Set signal.
		THIS^.signal.yellow.enable := TRUE;
		THIS^.signal.yellow.blink := TRUE;
		
		IF THIS^.inError() THEN
			// Reset drives.
			FOR iCounter := 1 TO 6 BY 1 DO
				Axis[iCounter].doReset();
			END_FOR
		ELSE
			// Enable drives if not enabled yet.
			IF NOT THIS^.isEnabled() THEN
				FOR iCounter := 1 TO 6 BY 1 DO
					Axis[iCounter].enabled := TRUE;
				END_FOR
			END_IF
			
			IF THIS^.isEnabled() THEN
				IF NOT bToggle THEN
					// Move pistons to home position.
					THIS^.goHomePosition();
					bToggle := TRUE;
				ELSE
					IF THIS^.isReady() THEN
						// When position has been reached go to stopped state.
						bToggle := FALSE;
						THIS^.state := stateFlightSimulator.stopped;
					END_IF
				END_IF
			END_IF
		END_IF
END_CASE

// Cycle Axis classes.
FOR iCounter := 1 TO 6 BY 1 DO
	THIS^.axis[iCounter].cycle();
END_FOR
// Cycle signal class.
THIS^.signal.cycle();
END_METHOD

METHOD goNeutralPosition : BOOL
VAR
	// Counter to cycle through axis.
	iCounter: INT;
END_VAR
IF THIS^.isReady() THEN
	FOR iCounter := 1 TO 6 BY 1 DO
		THIS^.axis[iCounter].doMovement(position := 200, velocity := 25, continuousUpdate:=FALSE);
	END_FOR
END_IF
END_METHOD

METHOD isReady : BOOL
VAR_INPUT
END_VAR
VAR
	// Counter to cycle through axis.
	iCounter: INT;
END_VAR
// Check ready status of all axis, when one is not ready return with FALSE.
FOR iCounter := 1 TO 6 BY 1 DO
	IF NOT THIS^.axis[iCounter].isReady() THEN
		isReady := FALSE;
		RETURN;
	END_IF;
END_FOR;

isReady := TRUE;
END_METHOD

METHOD doMovement : BOOL
VAR_INPUT
	positions : ARRAY[1..6] OF REAL;
	speeds : ARRAY[1..6] OF REAL;
END_VAR
VAR
	// Counter to cycle through axis.
	iCounter: INT;
	// Var that says its safe to execute this command, will be lowered in the FOR loop check.
	bSafe: BOOL := TRUE;
END_VAR
FOR iCounter := 1 TO 6 BY 1 DO
	// If any of the positions are larger than 390 or smaller than 10 don't execute the command.
	IF positions[iCounter] > 390 OR positions[iCounter] < 10 THEN
		bSafe := FALSE;
	END_IF
	
	// If any of the velocities are larger than 401 or smaller than 0 don't execute the command.
	IF speeds[iCounter] >= 401 OR speeds[iCounter] < 0 THEN
		bSafe := FALSE;
	END_IF
END_FOR

IF bSafe THEN
    FOR iCounter := 1 TO 6 BY 1 DO
        IF positions[iCounter] > 390 THEN
            Axis[iCounter].doMovement(position:=390, velocity:=speeds[iCounter], continuousUpdate:=FALSE);
        ELSIF positions[iCounter] < 10 THEN
            Axis[iCounter].doMovement(position:=100, velocity:=speeds[iCounter], continuousUpdate:=FALSE);
        ELSE
            Axis[iCounter].doMovement(position:=positions[iCounter], velocity:=speeds[iCounter], continuousUpdate:=TRUE);
        END_IF
    END_FOR
END_IF
END_METHOD

METHOD isInitialised : BOOL
VAR_INPUT
END_VAR
VAR
	// Counter to cycle through axis.
	iCounter: INT;
END_VAR
// Check if all axis are initialised, when one is not initialised return with FALSE.
FOR iCounter := 1 TO 6 BY 1 DO
	IF NOT THIS^.axis[iCounter].isInitialised() THEN
		isInitialised := FALSE;
		RETURN;
	END_IF;
END_FOR;

isInitialised := TRUE;
END_METHOD

METHOD init : BOOL
VAR_INPUT
	axis1: REFERENCE TO AXIS_REF_FESTO;
	axis2: REFERENCE TO AXIS_REF_FESTO;
	axis3: REFERENCE TO AXIS_REF_FESTO;
	axis4: REFERENCE TO AXIS_REF_FESTO;
	axis5: REFERENCE TO AXIS_REF_FESTO;
	axis6: REFERENCE TO AXIS_REF_FESTO;
	lightRed: REFERENCE TO BOOL;
	lightYellow: REFERENCE TO BOOL;
	lightGreen: REFERENCE TO BOOL;
	enabled: REFERENCE TO BOOL;
	// When this variable is HIGH it means that the safety system is active.
	// This means none of it's safety systems has been triggered.
	safetySystem: REFERENCE TO BOOL;
	newPositions: REFERENCE TO ARRAY[1..6] OF REAL;
	newVelocities: REFERENCE TO ARRAY[1..6] OF REAL;
END_VAR
THIS^.axis[1].init(axis1);
THIS^.axis[2].init(axis2);
THIS^.axis[3].init(axis3);
THIS^.axis[4].init(axis4);
THIS^.axis[5].init(axis5);
THIS^.axis[6].init(axis6);

THIS^.signal.init(lightRed, lightYellow, lightGreen);

THIS^.enabled REF= enabled;
THIS^.safetySystem REF= safetySystem;

THIS^.newPositions REF= newPositions;
THIS^.newVelocities REF= newVelocities;
END_METHOD

METHOD inError : BOOL
VAR
	// Counter to cycle through axis.
	iCounter: INT;
END_VAR
// Check error status of all axis, when one is in error return with TRUE.
FOR iCounter := 1 TO 6 BY 1 DO
	IF THIS^.axis[iCounter].inError() THEN
		inError := TRUE;
		RETURN;
	END_IF;
END_FOR;

InError := FALSE;
END_METHOD

METHOD goHomePosition : BOOL
VAR
	// Counter to cycle through axis.
	iCounter: INT;
END_VAR
// Abort current movement action.
FOR iCounter := 1 TO 6 BY 1 DO
	THIS^.axis[iCounter].doAbort();
END_FOR

IF THIS^.isReady() THEN
	FOR iCounter := 1 TO 6 BY 1 DO
		THIS^.axis[iCounter].doMovement(position := 10, velocity := 25, continuousUpdate:=FALSE);
	END_FOR
END_IF
END_METHOD

METHOD goTopPosition : BOOL
VAR
	// Counter to cycle through axis.
	iCounter: INT;
END_VAR
// Abort current movement action.
FOR iCounter := 1 TO 6 BY 1 DO
	THIS^.axis[iCounter].doAbort();
END_FOR

IF THIS^.isReady() THEN
	FOR iCounter := 1 TO 6 BY 1 DO
		THIS^.axis[iCounter].doMovement(position := 390, velocity := 25, continuousUpdate:=FALSE);
	END_FOR
END_IF
END_METHOD

METHOD PPState : stateFlightSimulator
PPState := THIS^.state;
END_METHOD

END_FUNCTION_BLOCK

// signal
FUNCTION_BLOCK signal
VAR_INPUT
	// Red light.
	red: light;
	// Yellow light.
	yellow: light;
	// Green light.
	green: light;
END_VAR
VAR
	
	// TON.
	clockTON: TON;
	// TOF.
	clockTOF: TOF;
	// Current clock state.
	clock: BOOL;
END_VAR

METHOD init : BOOL
VAR_INPUT
	red: REFERENCE TO BOOL;
	yellow: REFERENCE TO BOOL;
	green: REFERENCE TO BOOL;
END_VAR
VAR
END_VAR
THIS^.red.init(red, clock);
THIS^.yellow.init(yellow, clock);
THIS^.green.init(green, clock);
END_METHOD

METHOD cycle : BOOL
VAR_INPUT
END_VAR
clockTON(IN:= NOT clockTOF.Q, PT:=T#500MS);
clockTOF(IN:= clockTON.Q, PT:=T#500MS);
THIS^.clock := clockTOF.Q;

// Cycle light objects.
THIS^.red.cycle();
THIS^.yellow.cycle();
THIS^.green.cycle();
END_METHOD

END_FUNCTION_BLOCK

// Light
FUNCTION_BLOCK Light
VAR
	light: REFERENCE TO BOOL;
	clock: REFERENCE TO BOOL;
	
	enabled: BOOL := FALSE;
	blinking: BOOL := FALSE;
END_VAR

PROPERTY blink : BOOL
SET
THIS^.blinking := blink;
END_SET
GET
blink := THIS^.blinking;
END_GET
END_PROPERTY

METHOD init : BOOL
VAR_INPUT
	light: REFERENCE TO BOOL;
	clock: REFERENCE TO BOOL;
END_VAR
VAR
END_VAR
THIS^.light REF= light;
THIS^.clock REF= clock;
END_METHOD

METHOD cycle : BOOL
VAR_INPUT
END_VAR
IF THIS^.enabled THEN
	IF THIS^.blinking THEN
		// If blinking is enabled, turn light on or off depending on clock state.
		IF THIS^.clock THEN
			THIS^.light := TRUE;
		ELSE
			THIS^.light := FALSE;
		END_IF
	ELSE
			THIS^.light := TRUE;
	END_IF
ELSE
	THIS^.light := FALSE;
END_IF
END_METHOD

PROPERTY enable : BOOL
GET
enable := THIS^.enabled;
END_GET
SET
THIS^.enabled := enable;
END_SET
END_PROPERTY

END_FUNCTION_BLOCK

// PLC/Application/TcpClient
PROGRAM TcpClient
VAR

    // Client object that connects to client machine.
	fbTcpClient   : NBS.TCP_Client;
    // Read object that reads incomming data from client machine.
	fbTcpRead     : NBS.TCP_Read;
    // Write object that writes data to client machine.
	fbTcpWrite    : NBS.TCP_Write;
	
	sendLength : INT;
	
	// TON object for reset delay.
	tonResetDelay: TON;
	// Received telegram from Read object.
	received      : STRING(gvlSetting.gc_wMaxTelegram);
	// Sent telegram to Write object.
	sent          : STRING(4095);
	// JSON Parser object to parse read data.
	parseJSON     : JSON_TO_STRUCT;
	// JSON Composer object to compose data to write.
	composeJSON   : STRUCT_TO_JSON;
	// Struct that stores the received data in usable arrays.
	servoData     : ServoData;
    // Make connection.
	xConnect      : BOOL := TRUE;
	// Do composing.
	xCompose: BOOL;
	// Do write action.
	xWrite: BOOL;
	// Do parsing
	xParse: BOOL;
	
	j : INT := 1;
 
    // Do read action.
	xRead         : BOOL;
    // Size of read data telegram.
	udiRead       : UDINT;
	// Timeout in µs.
	udiTimeOut: UDINT := 500000;
	
	
	udiVal        : UDINT;
    pudiVal       : POINTER TO BYTE;
    iIndex        : INT;
	xMissingAck   : BOOL;
    udiResult     : UDINT;
    udiLastAck    : UDINT;
    udiNow        : UDINT;
    diagnosticSendTimer : TON;
    diagnosticBuildErrors : UDINT;
    cspReceiver : CSP_Receive;
END_VAR

 fbTcpClient(xEnable := xConnect, ipAddr := gvlSetting.gc_stIpAddr, uiPort := gvlSetting.gc_uiPort, udiTimeOut := udiTimeOut);
// 
// // Run when connection is active.
// IF fbTcpClient.xActive AND GVL.FlightSimulator.isInitialised() THEN
// 	
// 	IF fbTcpWrite.xDone THEN
// 		xWrite := FALSE;
// 	ELSIF NOT fbTcpWrite.xBusy THEN
// 		IF composeJSON.Done AND composeJSON.Execute THEN
// 			xCompose := FALSE;
// 			xWrite := TRUE;
// 		ELSIF (NOT composeJSON.Busy) THEN
// 			   xCompose := TRUE;
// 			   xWrite := FALSE;
// 		END_IF
// 	END_IF
// 	
// 	composeJSON(
// 		Execute:= xCompose,
// 		JSONString:= ADR(sent),
// 		JSONStringSize:= SIZEOF(sent),
// 		JSONVars:= ADR(GVL.currentPositions),
// 		NumberOfVars:= SIZEOF(GVL.currentPositions) / SIZEOF(JSONVAR)
// 	); 
// 	fbTcpWrite(xExecute := xWrite, hConnection := fbTcpClient.hConnection, udiTimeOut := udiTimeOut, szSize := SIZEOF(sent), pData := ADR(sent));
// 	
// 	IF (NOT fbTcpRead.xBusy) AND (NOT parseJSON.Busy) THEN
// 		xRead := TRUE;
// 	ELSIF fbTcpRead.xReady THEN
// 		xRead := FALSE;
// 		xParse := TRUE;
// 	ELSIF (NOT parseJSON.Busy) THEN
// 		xParse := FALSE;
// 	END_IF
// 
// 	parseJSON(
// 		Execute := xParse,
// 		JSONString:= ADR(received),
// 		JSONStringSize:= SIZEOF(received),
// 		JSONVars:= ADR(servoData),
// 		NumberOfVars:= SIZEOF(servoData) / SIZEOF(JSONVAR)
// 	);
// 	
// 	received := '';
// 	//FOR j := 1 TO SIZEOF(received) DO
// 	//	received[j] := 0;
// 	//END_FOR
// 	//sent := '';
// 	fbTcpRead(xEnable := xRead, hConnection := fbTcpClient.hConnection, szSize := SIZEOF(received), pData := ADR(received), szCount => udiRead);
// 	
// END_IF
// 
// // Reset connection when connection has stopped.
// IF (NOT xConnect) THEN
// 	// Reset all variables.
// 	xConnect := FALSE;
// 	xWrite := FALSE;
// 	xCompose := FALSE;
// 	fbTcpWrite(xExecute := FALSE);
// 	xRead := FALSE;
// 	xParse := FALSE;
// 	fbTcpRead(xEnable := FALSE);
// 	received := '';
// 	sent := '';
// 	// Delay reset for 3 sec.
// 	tonResetDelay(IN:=TRUE, PT:=T#3S);
// 	IF (tonResetDelay.Q) THEN
// 		tonResetDelay(IN:=FALSE);
// 		xConnect := TRUE;
// 	END_IF
// 	
// END_IF
// 
// IF fbTcpClient.xDone AND xConnect THEN
// 	xConnect := FALSE;
// END_IF
// 
// // Stop connection when in error.
// //IF fbTcpClient.xError OR fbTcpWrite.xError OR fbTcpRead.xError THEN
// IF fbTcpClient.xError OR fbTcpRead.xError THEN
// 
// 	xConnect := FALSE;
// 	fbTcpWrite(xExecute := FALSE);
// END_IF 
// 

// Run when connection is active.
//IF fbTcpClient.xActive AND GVL.FlightSimulator.isInitialised() THEN
IF fbTcpClient.xActive THEN
    IF CSP_Config.ControlMode <> CSP_Config.CONTROL_MODE_CSP THEN DriveDiagnostics(); END_IF
    diagnosticSendTimer(IN := NOT xWrite, PT := T#50MS);
    IF fbTcpWrite.xDone OR fbTcpWrite.xError THEN
        xWrite := FALSE;
    ELSIF NOT fbTcpWrite.xBusy AND diagnosticSendTimer.Q THEN
        IF CSP_Config.ControlMode = CSP_Config.CONTROL_MODE_CSP THEN sent := CSP_Feedback();
        ELSE sent := BuildDiagnosticFeedback(); END_IF
		sendLength := LongStringLength(pText := ADR(sent), maxLength := 4095);
		xWrite := sendLength > 0;
        IF NOT xWrite THEN diagnosticBuildErrors := diagnosticBuildErrors + 1; END_IF
    END_IF
    // Buffer remains unchanged while TCP_Write is busy. Send only meaningful
    // bytes (including the newline), never the unused NUL-filled capacity.
    fbTcpWrite(xExecute := xWrite, hConnection := fbTcpClient.hConnection, udiTimeOut := udiTimeOut,
    	szSize := INT_TO_UDINT(sendLength), pData := ADR(sent));

    IF CSP_Config.ControlMode <> CSP_Config.CONTROL_MODE_CSP THEN
    // -------------------------
    //  ONTVANGEN VAN STUARTSERVER
    // -------------------------
    IF (NOT fbTcpRead.xBusy) AND (NOT parseJSON.Busy) THEN
        xRead := TRUE;
    ELSIF fbTcpRead.xReady THEN
        xRead := FALSE;
        xParse := TRUE;
    ELSIF (NOT parseJSON.Busy) THEN
        xParse := FALSE;
    END_IF

    // A CSP endpoint must never be interpreted as a legacy PP step.
    IF FIND(received, '"controlMode"') > 0 THEN xParse := FALSE; received := ''; END_IF
    parseJSON(
        Execute         := xParse,
        JSONString      := ADR(received),
        JSONStringSize  := SIZEOF(received),
        JSONVars        := ADR(servoData),
        NumberOfVars    := SIZEOF(servoData) / SIZEOF(JSONVAR)
    );

    // Buffer leegmaken voor volgende receive
    received := '';
    fbTcpRead(
        xEnable    := xRead,
        hConnection:= fbTcpClient.hConnection,
        szSize     := SIZEOF(received),
        pData      := ADR(received),
        szCount    => udiRead
    );

    END_IF

END_IF


// Reset connection when connection has stopped.
 IF (NOT xConnect) THEN
 	// Reset all variables.
 	xConnect := FALSE;
 	xWrite := FALSE;
 	xCompose := FALSE;
	fbTcpWrite(xExecute := FALSE);
 	xRead := FALSE;
 	xParse := FALSE;
 	fbTcpRead(xEnable := FALSE);
	received := '';
 	sent := '';
 	// Delay reset for 3 sec.
 	tonResetDelay(IN:=TRUE, PT:=T#3S);
 	IF (tonResetDelay.Q) THEN
 		tonResetDelay(IN:=FALSE);
 		xConnect := TRUE;
 	END_IF
	
 END_IF
 
 IF fbTcpClient.xDone AND xConnect THEN
 	xConnect := FALSE;
 END_IF

 // Stop connection when in error.
 //IF fbTcpClient.xError OR fbTcpWrite.xError OR fbTcpRead.xError THEN
IF fbTcpClient.xError OR fbTcpRead.xError THEN

	xConnect := FALSE;
	fbTcpWrite(xExecute := FALSE);
END_IF 
IF CSP_Config.ControlMode = CSP_Config.CONTROL_MODE_CSP THEN
    cspReceiver(Connected:=fbTcpClient.xActive AND xConnect,Connection:=fbTcpClient.hConnection);
    IF cspReceiver.Error THEN xConnect := FALSE; END_IF
END_IF

END_PROGRAM

// PLC/Application/DriveDiagnostics
PROGRAM DriveDiagnostics
VAR_INPUT
    // The packet builder consumes these flags only after assembling a complete
    // message. Inputs permit that explicit handoff between CODESYS programs.
    targetNew : ARRAY[1..6] OF BOOL;
    followingNew : ARRAY[1..6] OF BOOL;
    sampleSequence : UDINT;
END_VAR
VAR
    // Passive readers only. No command, enable, reset, or axis configuration writes.
    positionReaders : ARRAY[1..6] OF MC_ReadActualPosition_Festo;
    velocityReaders : ARRAY[1..6] OF MC_ReadActualVelocity_Festo;
    parameterReader : MC_ReadParameter_Festo;
    actualPositions : ARRAY[1..6] OF REAL;
    actualVelocities : ARRAY[1..6] OF REAL;
    positionValid : ARRAY[1..6] OF BOOL;
    velocityValid : ARRAY[1..6] OF BOOL;
    driveTargets : ARRAY[1..6] OF LREAL;
    followingErrors : ARRAY[1..6] OF LREAL;
    targetTick : ARRAY[1..6] OF UDINT;
    followingTick : ARRAY[1..6] OF UDINT;
    readErrors : ARRAY[1..6] OF WORD;
    readErrorCount : UDINT;
    sampleTick : UDINT;
    pollAxis : INT := 1;
    pollFollowing : BOOL;
    pollActive : BOOL;
    pollReset : BOOL;
    pollInterval : TON;
    pollTimeout : TON;
    parameter : UINT;
    drive : REFERENCE TO AXIS_REF_FESTO;
    i : INT;
END_VAR

// User units are supplied by the Festo library. Valid AND NOT Error is required;
// never turn a failed read into a plausible zero-valued measurement.
positionReaders[1](Axis := servo_drive_1, Enable := TRUE);
positionReaders[2](Axis := servo_drive_2, Enable := TRUE);
positionReaders[3](Axis := servo_drive_3, Enable := TRUE);
positionReaders[4](Axis := servo_drive_4, Enable := TRUE);
positionReaders[5](Axis := servo_drive_5, Enable := TRUE);
positionReaders[6](Axis := servo_drive_6, Enable := TRUE);
velocityReaders[1](Axis := servo_drive_1, Enable := TRUE);
velocityReaders[2](Axis := servo_drive_2, Enable := TRUE);
velocityReaders[3](Axis := servo_drive_3, Enable := TRUE);
velocityReaders[4](Axis := servo_drive_4, Enable := TRUE);
velocityReaders[5](Axis := servo_drive_5, Enable := TRUE);
velocityReaders[6](Axis := servo_drive_6, Enable := TRUE);
sampleTick := TIME_TO_UDINT(TIME());
FOR i := 1 TO 6 DO
    positionValid[i] := positionReaders[i].Valid AND NOT positionReaders[i].Error;
    velocityValid[i] := velocityReaders[i].Valid AND NOT velocityReaders[i].Error;
    actualPositions[i] := positionReaders[i].Position;
    actualVelocities[i] := velocityReaders[i].Velocity;
END_FOR

// Only one SDO request is active across all six drives. Each request is followed
// by a 50 ms idle interval. Register traces are slower than the 20 Hz PDO traces.
// Do not increase this rate without measuring the actual fieldbus load.
CASE pollAxis OF
    1: drive REF= servo_drive_1;
    2: drive REF= servo_drive_2;
    3: drive REF= servo_drive_3;
    4: drive REF= servo_drive_4;
    5: drive REF= servo_drive_5;
    6: drive REF= servo_drive_6;
END_CASE
IF pollFollowing THEN parameter := 16#60F4; ELSE parameter := 16#607A; END_IF
IF pollReset THEN
    parameterReader(Axis := drive, Enable := FALSE);
    pollTimeout(IN := FALSE);
    pollInterval(IN := FALSE);
    pollReset := FALSE;
    IF pollFollowing THEN
        pollAxis := pollAxis + 1;
        IF pollAxis > 6 THEN pollAxis := 1; END_IF
    END_IF
    pollFollowing := NOT pollFollowing;
ELSE
    pollInterval(IN := NOT pollActive, PT := T#50MS);
    IF pollInterval.Q THEN pollActive := TRUE; END_IF
    parameterReader(Axis := drive, Enable := pollActive,
        ParameterNumber := parameter, SubindexNumber := 0);
    pollTimeout(IN := pollActive, PT := T#1S);
    IF pollActive AND (parameterReader.Valid OR parameterReader.Error OR pollTimeout.Q) THEN
        IF parameterReader.Valid AND NOT parameterReader.Error THEN
            IF pollFollowing THEN
                followingErrors[pollAxis] := parameterReader.Value;
                followingTick[pollAxis] := sampleTick;
                followingNew[pollAxis] := TRUE;
            ELSE
                driveTargets[pollAxis] := parameterReader.Value;
                targetTick[pollAxis] := sampleTick;
                targetNew[pollAxis] := TRUE;
            END_IF
            readErrors[pollAxis] := 0;
        ELSE
            readErrorCount := readErrorCount + 1;
            IF pollTimeout.Q THEN readErrors[pollAxis] := 16#FFFF;
            ELSE readErrors[pollAxis] := parameterReader.ErrorID; END_IF
            IF pollFollowing THEN followingNew[pollAxis] := FALSE;
            ELSE targetNew[pollAxis] := FALSE; END_IF
        END_IF
        pollActive := FALSE;
        pollReset := TRUE;
    END_IF
END_IF

END_PROGRAM

// PLC/Application/CSP_Feedback
FUNCTION CSP_Feedback : STRING(4095)
VAR
    output : STRING(4095);
    fragment : STRING(255);
    i, field : INT;
    ok : BOOL;
    cycle : UDINT;
    snapshot : ARRAY[1..6] OF CSP_AxisData;
END_VAR

cycle := CSP_Data.CycleCounter;
snapshot := CSP_Data.Axis;
IF cycle <> CSP_Data.CycleCounter THEN CSP_Feedback := ''; RETURN; END_IF
FOR i := 1 TO 6 DO
    IF NOT snapshot[i].Ready THEN CSP_Feedback := ''; RETURN; END_IF
END_FOR
output := '{"currentPositions":['; ok := TRUE;
FOR i := 1 TO 6 DO
    IF i > 1 THEN ok := AppendDiagnosticText(',',output) AND ok; END_IF
    ok := AppendDiagnosticText(LREAL_TO_STRING(snapshot[i].ActualPosition),output) AND ok;
END_FOR
ok := AppendDiagnosticText('],"diagnostics":{"version":2,"controlMode":8,"positionUnit":"mm","velocityUnit":"mm/s","registerUnit":"raw CiA402","targetSource":"CSP PDO command","followingErrorSource":"0x60F4 PDO","plcTickMs":',output) AND ok;
ok := AppendDiagnosticText(UDINT_TO_STRING(TIME_TO_UDINT(TIME())),output) AND ok;
FOR field := 1 TO 14 DO
    CASE field OF
        1: fragment := ',"receivedPositions":[';
        2: fragment := ',"receivedSpeeds":[';
        3: fragment := ',"actualPositions":[';
        4: fragment := ',"actualVelocities":[';
        5: fragment := ',"driveTargetPositions":[';
        6: fragment := ',"followingErrors":[';
        7: fragment := ',"commandPositions":[';
        8: fragment := ',"commandVelocities":[';
        9: fragment := ',"commandAccelerations":[';
        10: fragment := ',"modeRequested":[';
        11: fragment := ',"modeActual":[';
        12: fragment := ',"cia402State":[';
        13: fragment := ',"positionLimit":[';
        14: fragment := ',"communicationTimeout":[';
    END_CASE
    ok := AppendDiagnosticText(fragment,output) AND ok;
    FOR i := 1 TO 6 DO
        IF i > 1 THEN ok := AppendDiagnosticText(',',output) AND ok; END_IF
        CASE field OF
            1: fragment := LREAL_TO_STRING(snapshot[i].RequestedPosition);
            2: fragment := '0';
            3: fragment := LREAL_TO_STRING(snapshot[i].ActualPosition);
            4: fragment := LREAL_TO_STRING(snapshot[i].ActualVelocity);
            5: fragment := DINT_TO_STRING(snapshot[i].TargetRaw);
            6: fragment := DINT_TO_STRING(snapshot[i].FollowingErrorRaw);
            7: fragment := LREAL_TO_STRING(snapshot[i].CommandPosition);
            8: fragment := LREAL_TO_STRING(snapshot[i].CommandVelocity);
            9: fragment := LREAL_TO_STRING(snapshot[i].CommandAcceleration);
            10: fragment := SINT_TO_STRING(snapshot[i].ModeRequested);
            11: fragment := SINT_TO_STRING(snapshot[i].ModeActual);
            12: fragment := UINT_TO_STRING(WORD_TO_UINT(snapshot[i].CiA402State));
            13: fragment := INT_TO_STRING(BOOL_TO_INT(snapshot[i].PositionLimit));
            14: fragment := INT_TO_STRING(BOOL_TO_INT(snapshot[i].CommunicationTimeout));
        END_CASE
        IF field >= 7 AND field <= 9 AND NOT CSP_Data.Active THEN fragment := 'null'; END_IF
        ok := AppendDiagnosticText(fragment,output) AND ok;
    END_FOR
    ok := AppendDiagnosticText(']',output) AND ok;
END_FOR
ok := AppendDiagnosticText(',"resetRequired":',output) AND ok;
ok := AppendDiagnosticText(INT_TO_STRING(BOOL_TO_INT(CSP_Data.ResetRequired)),output) AND ok;
ok := AppendDiagnosticText(',"homing":',output) AND ok;
ok := AppendDiagnosticText(INT_TO_STRING(BOOL_TO_INT(CSP_Data.Homing)),output) AND ok;
ok := AppendDiagnosticText(',"readyToStart":',output) AND ok;
ok := AppendDiagnosticText(INT_TO_STRING(BOOL_TO_INT(CSP_Data.ReadyToStart)),output) AND ok;
ok := AppendDiagnosticText('}}$N',output) AND ok;
// Build the packet from the coherent copy, outside the EtherCAT task.
IF ok THEN CSP_Feedback := output; ELSE CSP_Feedback := ''; END_IF

END_FUNCTION

// PLC/Application/AppendDiagnosticText
FUNCTION AppendDiagnosticText : BOOL
VAR_INPUT
    fragment : STRING(255);
END_VAR
VAR_IN_OUT
    destination : STRING(4095);
END_VAR
VAR
    used : INT;
    count : INT;
    i : INT;
    outputBytes : POINTER TO BYTE;
    inputBytes : POINTER TO BYTE;
END_VAR

